METHOD M_Run
CASE _step OF
    0:
        M_Step(StepNo := 10, StepName := 'project.test.raiseIdle', Awaits := 0,
            AwaitingLabel := '', TimeClass := E_TimeClass.WORK, ExpectedTime := T#0S);
        _retVal := E_StepResult.ADVANCE;
        M_Advance(OnAdvance := 20);
    20:  // conditional command. `Enable` decides whether the child is driven at all,
         // so this step cannot hand it to the §6.9 auto-rollup - Awaits would name a
         // module it may never command. M_RaiseFromChild adopts the child's own
         // first-out instead, verbatim, with the child as the §3.13 drill-down link.
        M_Step(StepNo := 20, StepName := 'project.test.raiseCommand', Awaits := 0,
            AwaitingLabel := '', TimeClass := E_TimeClass.WORK, ExpectedTime := T#0S);
        IF ReportOnly THEN
            // The step already routes the failure itself, so it PUBLISHES the child's
            // first-out and carries on - the §6.9(e) counterpart of raising it.
            IF M_ReportFromChild(Source := _child) THEN
                _child.Execute := FALSE;
                _retVal := E_StepResult.ADVANCE;
            END_IF
        ELSIF M_RaiseFromChild(Source := _child) THEN
            _child.Execute := FALSE;         // §6.1 drop-reset frees the child to recover
            RETURN;                          // chain stopped; the Unit is in ERROR
        END_IF
        // §6.9(e) — called unconditionally every scan the step runs. The base
        // raises it ONCE per visit, so the ring gets one entry per occurrence and
        // the chain is never stopped by it.
        IF SimWarn THEN
            Warned := M_RaiseWarning(Reason := E_Reason.TEST_FAULT,
                DescriptionKey := 'project.test.stepWarning',
                Severity := E_Severity.LOW, Category := E_Category.PROCESS);
        END_IF
        IF Enable THEN
            IF M_TryIssue(Steppable := TRUE) THEN
                Issues := Issues + 1;        // proves the re-evaluation after resume
                _child.Abort := FALSE;
                _child.Execute := TRUE;
            END_IF
            IF _child.Done THEN
                _child.Execute := FALSE;
                _retVal := E_StepResult.ADVANCE;
            END_IF
        END_IF
        M_Advance(OnAdvance := 30);
    30:  // application rule: nothing in the framework can see it, so the step
         // defines the whole message - severity, category and drill-down link (§8.1).
        M_Step(StepNo := 30, StepName := 'project.test.raiseCustom', Awaits := 0,
            AwaitingLabel := '', TimeClass := E_TimeClass.WORK, ExpectedTime := T#0S);
        IF SimCustom THEN
            // A PROJECT BAND code (10000+), deliberately: M_RaiseCustom documents
            // that Severity/Category are a proposal the §8.8 rationalization
            // overrides for any REGISTERED reason, and every E_Reason member is
            // registered by construction (the catalog generator refuses one that
            // is not). Raising E_Reason.TEST_FAULT here therefore asserted the
            // opposite of what the test says it proves: the registry's LOW/SYSTEM
            // correctly replaced the step's HIGH/PROCESS. Only a band code the
            // registry does not know keeps the step's own choice.
            IF M_RaiseCustom(Reason := 10999,
                DescriptionKey := 'project.test.customRaise',
                Severity := E_Severity.HIGH, Category := E_Category.PROCESS,
                LinkPath := _child.Name) THEN
                RETURN;
            END_IF
        END_IF
        _retVal := E_StepResult.ADVANCE;
        M_Advance(OnAdvance := 999);
    999:
        M_Step(StepNo := 999, StepName := 'project.test.raiseComplete', Awaits := 0,
            AwaitingLabel := '', TimeClass := E_TimeClass.WORK, ExpectedTime := T#0S);
        Done := TRUE;
        M_Complete();
ELSE
    M_Fault(Reason := E_Reason.STEP_STALLED, DescriptionKey := 'std.error.undefinedStep');
END_CASE
END_METHOD

END_FUNCTION_BLOCK

// ---- Fraktal_Tests/FB_SequencePar_Tests.TcPOU
// Core §6.12 — parallel branches. Proves the three things that make them real
// rather than drawn: both legs run in the SAME scan with independent latches, the
// join waits for the slowest, and each leg is published as its own §3.13 rows.
FUNCTION_BLOCK FB_SequencePar_Tests EXTENDS TcUnit.FB_TestSuite
VAR
    _u : FB_ProbeUnitPar;
    _w1, _w2 : BOOL;
    _rowA, _rowB : INT;
    _i : INT;
END_VAR

Legs_run_together_with_independent_step_state();
Join_waits_for_every_leg_and_publishes_them_separately();

METHOD Legs_run_together_with_independent_step_state
TEST('Legs_run_together_with_independent_step_state');
IF NOT _w1 THEN
    AssertTrue(Condition := _u.Setup(Name := 'Test.Par'), Message := 'Unit sets up');
    AssertTrue(Condition := _u.Start(), Message := 'Unit starts');
    _u();                                // fork scan: BOTH legs run
    AssertEquals_UDINT(Expected := 1, Actual := _u.M_TestIssues(Leg := 1),
        Message := 'leg 1 issued its command');
    AssertEquals_UDINT(Expected := 1, Actual := _u.M_TestIssues(Leg := 2),
        Message := 'leg 2 issued its own command in the SAME scan - one shared issue latch used to let leg 1 consume the latch belonging to leg 2');
    _u();
    AssertEquals_UDINT(Expected := 1, Actual := _u.M_TestIssues(Leg := 1),
        Message := 'and neither re-issues while its step is still running (§6.1 one-shot, per leg)');
    _w1 := TRUE;
END_IF
TEST_FINISHED();
END_METHOD

METHOD Join_waits_for_every_leg_and_publishes_them_separately
TEST('Join_waits_for_every_leg_and_publishes_them_separately');
IF NOT _w2 THEN
    // both leg rows are live at once - the whole reason a single CurrentStep was
    // not enough to draw a parallel step (§3.13/§6.12)
    FOR _i := 1 TO _u.SequenceStepCount DO
        IF _u.SequenceStepDef[_i].StepNo = 600 THEN _rowA := _i; END_IF
        IF _u.SequenceStepDef[_i].StepNo = 700 THEN _rowB := _i; END_IF
    END_FOR
    AssertTrue(Condition := (_rowA > 0) AND (_rowB > 0),
        Message := 'each leg publishes its own rows, offset by its BaseStepNo');
    AssertEquals_INT(Expected := 1, Actual := _u.SequenceStepDef[_rowA].Branch,
        Message := 'tagged with the leg the fork assigned it');
    AssertEquals_INT(Expected := 2, Actual := _u.SequenceStepDef[_rowB].Branch,
        Message := 'and the other leg with its own');
    AssertTrue(Condition := (_u.ActiveSteps[1].RowIdx = _rowA)
        AND (_u.ActiveSteps[2].RowIdx = _rowB),
        Message := 'BOTH rows are active at the same time - one cursor per leg');
    // leg 1 finishes; the join must not fire on it alone
    _u.M_TestSetChild(Which := 1, ChildDone := TRUE);
    _u();                                // child A completes
    _u();                                // leg 1 advances to its terminal step
    _u();                                // leg 1 reports Done
    AssertEquals_INT(Expected := 500, Actual := _u.M_TestChainStep(),
        Message := 'the join holds the fork step while leg 2 is still working');
    AssertFalse(Condition := _u.Done, Message := 'and the Unit has not completed');
    _u.M_TestSetChild(Which := 2, ChildDone := TRUE);
    _u();                                // child B completes
    _u();                                // leg 2 advances
    _u();                                // leg 2 Done -> join fires
    _u();                                // chain reaches its completion step
    AssertEquals_INT(Expected := 999, Actual := _u.M_TestChainStep(),
        Message := 'the fork step commits only once EVERY leg is Done');
    _w2 := TRUE;
END_IF
TEST_FINISHED();
END_METHOD

END_FUNCTION_BLOCK

// ---- Fraktal_Tests/FB_ProbeUnitPar.TcPOU
// Unit host for the §6.12 parallel suite: two children, one forking chain.
FUNCTION_BLOCK FB_ProbeUnitPar EXTENDS FB_UnitBase
VAR
    ChildA : FB_ProbeCM;
    ChildB : FB_ProbeCM;
    Chain : FB_ProbeParChain;
END_VAR

Cyclic();

METHOD Setup : BOOL
VAR_INPUT
    Name : STRING(80);
END_VAR
_M_SetName(Name);
StallTime := T#10S;
Setup := ChildA.Setup(Name := CONCAT(Name, '.ChildA'))
    AND ChildB.Setup(Name := CONCAT(Name, '.ChildB'))
    AND _M_Register(Child := ChildA)
    AND _M_Register(Child := ChildB)
    AND Chain.Setup(Host := THIS^, ChildA := ChildA, ChildB := ChildB);
END_METHOD

METHOD PROTECTED OnCyclic : DINT
OnCyclic := SUPER^.OnCyclic();   // base first (Core §3.14.2)
_M_TickChildren();
END_METHOD

METHOD PROTECTED _M_Dispatch
Chain.M_Run();
END_METHOD

METHOD PROTECTED OnCommandStart : DINT
OnCommandStart := SUPER^.OnCommandStart();
Chain.M_Reset();
END_METHOD

METHOD M_TestSetChild : BOOL
VAR_INPUT
    Which : INT;
    ChildDone : BOOL;
END_VAR
IF Which = 1 THEN
    ChildA.SimDone := ChildDone;
ELSE
    ChildB.SimDone := ChildDone;
END_IF
M_TestSetChild := TRUE;
END_METHOD

METHOD M_TestIssues : UDINT
VAR_INPUT
    Leg : INT;
END_VAR
M_TestIssues := Chain.M_TestIssues(Leg := Leg);
END_METHOD

METHOD M_TestChainStep : INT
M_TestChainStep := Chain.ActiveStep;
END_METHOD

END_FUNCTION_BLOCK

// ---- Fraktal_Tests/FB_ProbeParChain.TcPOU
// §6.12 — the ST form of a parallel divergence: ONE fork step that runs each leg
// and joins on all of them. Two work positions running simultaneously and
// independently is exactly this shape, and it needs no chart.
FUNCTION_BLOCK FB_ProbeParChain EXTENDS FB_SequenceBase
VAR
    LegA : FB_ProbeLeg;
    LegB : FB_ProbeLeg;
END_VAR

;

METHOD Setup : BOOL
VAR_INPUT
    Host : I_SequenceHost;
END_VAR
VAR_IN_OUT
    ChildA : FB_ProbeCM;
    ChildB : FB_ProbeCM;
END_VAR
Setup := M_Attach(Host := Host)
    AND LegA.Setup(Host := Host, Child := ChildA)
    AND LegB.Setup(Host := Host, Child := ChildB);
END_METHOD

METHOD M_Reset
M_ResetBase(FirstStep := 0);
END_METHOD

METHOD M_Run
CASE _step OF
    0:  // the fork. One M_RunPar per leg, one M_ParJoin: the leg list is the calls
        // themselves, so there is nothing to register and nothing to keep in step
        // when a leg is added or removed (§1.1 O1).
        M_Step(StepNo := 500, StepName := 'project.test.forkBothPositions', Awaits := 0,
            AwaitingLabel := '', TimeClass := E_TimeClass.WORK, ExpectedTime := T#0S);
        M_RunPar(Chain := LegA, BaseStepNo := 600, Branch := 1);
        M_RunPar(Chain := LegB, BaseStepNo := 700, Branch := 2);
        _retVal := M_ParJoin();
        M_Advance(OnAdvance := 999);
    999:
        M_Step(StepNo := 999, StepName := 'project.test.parallelComplete', Awaits := 0,
            AwaitingLabel := '', TimeClass := E_TimeClass.WORK, ExpectedTime := T#0S);
        Done := TRUE;
        M_Complete();
ELSE
    M_Fault(Reason := E_Reason.STEP_STALLED, DescriptionKey := 'std.error.undefinedStep');
END_CASE
END_METHOD

// test seam: how many times each leg issued its own command
METHOD M_TestIssues : UDINT
VAR_INPUT
    Leg : INT;
END_VAR
IF Leg = 1 THEN
    M_TestIssues := LegA.Issues;
ELSE
    M_TestIssues := LegB.Issues;
END_IF
END_METHOD

END_FUNCTION_BLOCK

// ---- Fraktal_Tests/FB_ProbeLeg.TcPOU
// §6.12 — one leg of a parallel step, written as an ORDINARY chain. That is the
// whole point of the ST form: a leg is a chain, so it brings its own step pointer,
// its own transition result and its own step-scoped latches, and nothing about it
// has to know it is running beside another one.
FUNCTION_BLOCK FB_ProbeLeg EXTENDS FB_SequenceBase
VAR_OUTPUT
    Issues : UDINT;                    // times this leg issued its command
END_VAR
VAR
    {attribute 'OPC.UA.DA' := '0'}
    _child : REFERENCE TO FB_ProbeCM;
END_VAR

;

METHOD Setup : BOOL
VAR_INPUT
    Host : I_SequenceHost;
END_VAR
VAR_IN_OUT
    Child : FB_ProbeCM;
END_VAR
_child REF= Child;
Setup := M_Attach(Host := Host) AND __ISVALIDREF(_child);
END_METHOD

METHOD PROTECTED OnChainReset
Issues := 0;
END_METHOD

// Run as a composite/parallel leg, so the step records are offset by _baseStepNo
// (§6.5) and the chart still reads as one continuous chain.
METHOD M_ChainRun
CASE _step OF
    0:
        M_Step(StepNo := _baseStepNo, StepName := 'project.test.legCommand', Awaits := 0,
            AwaitingLabel := '', TimeClass := E_TimeClass.WORK, ExpectedTime := T#0S);
        IF M_TryIssue(Steppable := TRUE) THEN
            Issues := Issues + 1;
            _child.Abort := FALSE;
            _child.Execute := TRUE;
        END_IF
        IF _child.Done THEN
            _child.Execute := FALSE;
            _retVal := E_StepResult.ADVANCE;
        END_IF
        M_Advance(OnAdvance := 999);
    999:
        M_Step(StepNo := _baseStepNo + 90, StepName := 'project.test.legDone', Awaits := 0,
            AwaitingLabel := '', TimeClass := E_TimeClass.WORK, ExpectedTime := T#0S);
        Done := TRUE;                  // the join reads this
ELSE
    M_Fault(Reason := E_Reason.STEP_STALLED, DescriptionKey := 'std.error.undefinedStep');
END_CASE
END_METHOD

END_FUNCTION_BLOCK

// ---- Fraktal_Tests/FB_StateFlag_Tests.TcPOU
// Core §3.12 — derived state flags. The point of the mechanism is that a flag is
// a live fact, not a latch, so the tests are about what happens when the fact
// changes and when the module stops asserting it at all.
FUNCTION_BLOCK FB_StateFlag_Tests EXTENDS TcUnit.FB_TestSuite
VAR
    _m : FB_ProbeCM;
    _w1, _w2 : BOOL;
    _since : DT;
END_VAR

Flag_is_published_with_the_moment_it_changed();
Unpublished_flag_goes_stale_and_stops_claiming();

METHOD Flag_is_published_with_the_moment_it_changed
TEST('Flag_is_published_with_the_moment_it_changed');
IF NOT _w1 THEN
    AssertTrue(Condition := _m.Setup(Name := 'Test.State'), Message := 'module sets up');
    _m.SimState := TRUE;
    _m();
    AssertTrue(Condition := _m.StateProbe,
        Message := 'the call returns the value, so it reads as a plain assignment');
    AssertEquals_INT(Expected := 1, Actual := _m.StateFlagCount,
        Message := 'and publishes it on the generic table');
    AssertEquals_STRING(Expected := 'project.test.probeState',
        Actual := _m.StateFlags[1].Key, Message := 'under the key the module chose');
    AssertTrue(Condition := _m.StateFlags[1].Value, Message := 'with the value');
    AssertFalse(Condition := _m.StateFlags[1].Stale, Message := 'and not stale');
    _since := _m.StateFlags[1].Since;
    _m();
    AssertEquals_DWORD(Expected := DT_TO_DWORD(_since),
        Actual := DT_TO_DWORD(_m.StateFlags[1].Since),
        Message := 'Since is the moment it CHANGED, not the last time it was written');
    // the fact stops being true: a derived flag follows it with no sequence involved
    _m.SimState := FALSE;
    _m();
    AssertFalse(Condition := _m.StateFlags[1].Value,
        Message := 'a derived flag drops itself - this is what a latched OutCmd could not do');
    _w1 := TRUE;
END_IF
TEST_FINISHED();
END_METHOD

METHOD Unpublished_flag_goes_stale_and_stops_claiming
TEST('Unpublished_flag_goes_stale_and_stops_claiming');
IF NOT _w2 THEN
    _m.SimState := TRUE;
    _m();
    AssertTrue(Condition := _m.StateFlags[1].Value, Message := 'true again');
    // the project puts the publication behind a condition that stops being true
    _m.SimPublish := FALSE;
    _m();                                // last scan's publication still stands
    _m();                                // the sweep resolves it
    AssertTrue(Condition := _m.StateFlags[1].Stale,
        Message := 'a flag nobody computes any more is marked stale');
    AssertFalse(Condition := _m.StateFlags[1].Value,
        Message := 'and forced FALSE: unmaintained state is not a claim (§5.6)');
    _w2 := TRUE;
END_IF
TEST_FINISHED();
END_METHOD

END_FUNCTION_BLOCK

// ---- Fraktal_Tests/FB_Axis_Tests.TcPOU
// Annex G axis CM. T1/T4 are proven once in FB_Base_Tests and not repeated (S5.7).
//
// SCOPE, stated plainly: this host has no NC PTP licence, so no test here moves a
// real axis. Every test below asserts behaviour that occurs BEFORE any MC_* call
// is issued - request validation, the ownership contract, and the handshake. The
// MC_* interaction itself is unproven and recorded as such in the evidence.
//
// That is also why _M_MoveTo validates the request (soft limits) before the state
// (homed): both rejections are provable without a drive, and reporting "not
// homed" for an impossible target would send an operator to the wrong problem.
FUNCTION_BLOCK FB_Axis_Tests EXTENDS TcUnit.FB_TestSuite
VAR
    _ax1 : AXIS_REF;
    _cm1 : FB_AxisCM;
    _ax2 : AXIS_REF;
    _cm2 : FB_AxisCM;
    _ax3 : AXIS_REF;
    _cm3 : FB_AxisCM;
    _ax4 : AXIS_REF;
    _cm4 : FB_AxisCM;
    _w1, _w2, _w3, _w4 : BOOL;
END_VAR

Library_declares_no_interlocks_and_the_application_owns_safe_motion_status();
Target_outside_soft_limits_is_rejected_before_any_motion();
Move_before_home_is_rejected();
Unsupported_command_is_rejected();

METHOD Library_declares_no_interlocks_and_the_application_owns_safe_motion_status
TEST('Library_declares_no_interlocks_and_the_application_owns_safe_motion_status');
IF NOT _w1 THEN
    _cm1.Setup(Name := 'Axis1', AxisRef := _ax1, Recipe := 0);
    _cm1();
    // S7.2.1 + S9.2: a library cannot name "STO cleared" for a station it has
    // never seen, so it declares nothing and the application supplies the
    // read-only safe-motion status it can see.
    AssertTrue(Condition := _cm1.Intlk.AllOk,
        Message := 'a library type that declares no interlock does not gate the axis');
    AssertTrue(Condition := _cm1.DeclareCondition(Index := 1,
            DescriptionKey := 'std.interlock.areaSafe',
            Reason := E_Reason.INTERLOCK_DROPPED, Bypassable := FALSE),
        Message := 'the application declares its own safe-motion condition');
    _cm1();
    AssertFalse(Condition := _cm1.Intlk.AllOk,
        Message := 'a declared but undriven condition is fail-closed');
    _cm1.SetCondition(Index := 1, Ok := TRUE);
    _cm1();
    AssertTrue(Condition := _cm1.Intlk.AllOk, Message := 'and clears once driven');
    _w1 := TRUE;
END_IF
TEST_FINISHED();
END_METHOD

METHOD Target_outside_soft_limits_is_rejected_before_any_motion
TEST('Target_outside_soft_limits_is_rejected_before_any_motion');
IF NOT _w2 THEN
    _cm2.Setup(Name := 'Axis2', AxisRef := _ax2, Recipe := 0);
    _cm2.ParCfg.SoftMin := 0.0;
    _cm2.ParCfg.SoftMax := 100.0;
    _cm2.ParCmd.Target := 150.0;                  // beyond SoftMax
    _cm2.Command := E_AxisCommand.MOVE_TO;
    _cm2.Execute := TRUE;
    _cm2(); _cm2();
    // S5.6: reject the malformed request rather than commanding motion and
    // discovering the problem at a limit switch.
    AssertTrue(Condition := _cm2.Error, Message := 'an out-of-range target is refused');
    AssertEquals_DWORD(Expected := TO_DWORD(PL_ModuleReasons.AXIS_TARGET_OOR),
        Actual := _cm2.ErrorID, Message := 'with AXIS_TARGET_OOR');
    AssertEquals_STRING(Expected := 'Axis2', Actual := _cm2.Status.Diagnostic.SourcePath,
        Message := 'and the module as its source path');
    _w2 := TRUE;
END_IF
TEST_FINISHED();
END_METHOD

METHOD Move_before_home_is_rejected
TEST('Move_before_home_is_rejected');
IF NOT _w3 THEN
    _cm3.Setup(Name := 'Axis3', AxisRef := _ax3, Recipe := 0);
    _cm3.ParCfg.SoftMin := 0.0;
    _cm3.ParCfg.SoftMax := 100.0;
    _cm3.ParCmd.Target := 50.0;                   // in range, but the axis is not homed
    _cm3.Command := E_AxisCommand.MOVE_TO;
    _cm3.Execute := TRUE;
    _cm3(); _cm3();
    AssertTrue(Condition := _cm3.Error, Message := 'a move before homing is refused');
    AssertEquals_DWORD(Expected := TO_DWORD(PL_ModuleReasons.AXIS_NOT_HOMED),
        Actual := _cm3.ErrorID, Message := 'with AXIS_NOT_HOMED');
    AssertFalse(Condition := _cm3.OutImm.Homed, Message := 'and the axis reports not homed');
    _w3 := TRUE;
END_IF
TEST_FINISHED();
END_METHOD

METHOD Unsupported_command_is_rejected
TEST('Unsupported_command_is_rejected');
IF NOT _w4 THEN
    _cm4.Setup(Name := 'Axis4', AxisRef := _ax4, Recipe := 0);
    _cm4.Command := E_AxisCommand.NONE;           // never a valid request (S5.6)
    _cm4.Execute := TRUE;
    _cm4(); _cm4();
    AssertTrue(Condition := _cm4.Error, Message := 'an unset command is refused');
    AssertEquals_DWORD(Expected := TO_DWORD(E_Reason.UNSUPPORTED_COMMAND),
        Actual := _cm4.ErrorID, Message := 'with UNSUPPORTED_COMMAND');
    _w4 := TRUE;
END_IF
TEST_FINISHED();
END_METHOD

END_FUNCTION_BLOCK

// ---- Fraktal_Tests/FB_RobotPlanner_Tests.TcPOU
// Annex I I.9-I.10.2 route planner, against the geometry of the reviewed cell.
//
// The fixture is deliberately the real thing rather than a toy: five help
// points, the twelve work positions of a plasma-clean handling cell, and the
// scan position that sits between two transit regions - reachable from the
// drawer side via HELP4 and the process side via HELP5. That junction is the
// case the reference framework could not express declaratively and hand-coded
// in two different methods from private state; if the affinity table cannot
// reproduce it in BOTH directions with no branching, the model has failed and
// it is better to find out here than in an annex.
//
// No arm, no connector, no motion: the planner is pure logic (S5.7, Annex H).
FUNCTION_BLOCK FB_RobotPlanner_Tests EXTENDS TcUnit.FB_TestSuite
VAR CONSTANT
    // helps
    HELP1 : INT := 1;   // change-position side
    HELP2 : INT := 2;   // left drawer
    HELP3 : INT := 3;   // home / NIO drawer
    HELP4 : INT := 4;   // drawer-side scan approach
    HELP5 : INT := 5;   // process side
    // nests
    CP_GRIPPER1    : INT := 1;
    READ_GRIPPER   : INT := 2;
    SCAN_PART      : INT := 3;
    DRAWER_LEFT    : INT := 4;
    DRAWER_RIGHT   : INT := 5;
    DRAWER_NIO     : INT := 6;
    PROCESS_START  : INT := 7;
    ONE_WAY_NEST   : INT := 8;   // synthetic: entry-only, to prove the loud refusal
    ISLAND_NEST    : INT := 9;   // synthetic: served by a help with no graph edge
    // transit regions
    REGION_DRAWER  : DWORD := 1;
    REGION_PROCESS : DWORD := 2;
    // grippers
    G_WITH : INT := 1;   // a gripper is coupled - tall approach
    G_NONE : INT := 2;   // nothing coupled - short approach
END_VAR
VAR
    _graph : ST_RouteGraph;
    _geom  : ST_RobotGeometry;
    _p     : FB_RobotRoutePlanner;
    _route : ST_RobotPointList;
    _ret   : DINT;
    _help  : INT;
    _built : BOOL;
    _w1, _w2, _w3, _w4, _w5, _w6, _w7, _w8, _w9, _w10 : BOOL;
END_VAR

IF NOT _built THEN
    _M_BuildFixture();
    _built := TRUE;
END_IF

Scan_junction_resolves_the_process_side_help();
Scan_junction_resolves_the_drawer_side_help_in_the_same_table();
Nest_to_nest_emits_depart_then_transit_then_approach();
Approach_corridor_is_reversed_and_lands_exactly_on_the_nest();
Corridor_differs_per_gripper_with_no_conditional_code();
Taught_corridor_emits_a_list_reference_instead_of_offsets();
Disconnected_graph_yields_ROBOT_NO_ROUTE();
One_way_nest_refuses_the_reversal_loudly();
Malformed_endpoints_are_rejected_before_planning();
Direct_nest_list_bypasses_help_routing();

// The reviewed cell as configuration - which is the whole point: a station
// supplies a table, not traversal code.
METHOD PRIVATE _M_BuildFixture
VAR
    _i : INT;
END_VAR
// --- help geometry and the transit graph -------------------------------
_geom.HelpPose[HELP1].X := 0;    _geom.HelpPose[HELP1].Z := 1000;
_geom.HelpPose[HELP2].X := 500;  _geom.HelpPose[HELP2].Z := 1000;
_geom.HelpPose[HELP3].X := 1000; _geom.HelpPose[HELP3].Z := 1000;
_geom.HelpPose[HELP4].X := 1500; _geom.HelpPose[HELP4].Z := 1000;
_geom.HelpPose[HELP5].X := 2000; _geom.HelpPose[HELP5].Z := 1000;

_graph.HelpRegion[HELP1] := REGION_DRAWER;
_graph.HelpRegion[HELP2] := REGION_DRAWER;
_graph.HelpRegion[HELP3] := REGION_DRAWER;
_graph.HelpRegion[HELP4] := REGION_DRAWER;
_graph.HelpRegion[HELP5] := REGION_PROCESS;

// a simple chain HELP1..HELP5, bidirectional
FOR _i := 1 TO 4 DO
    _graph.HelpAdj[_i, _i + 1] := TRUE;
    _graph.HelpAdj[_i + 1, _i] := TRUE;
END_FOR

// --- nest geometry -----------------------------------------------------
_geom.NestPose[G_WITH, DRAWER_LEFT].X  := 500;
_geom.NestPose[G_WITH, DRAWER_LEFT].Y  := 200;
_geom.NestPose[G_WITH, DRAWER_LEFT].Z  := 100;
_geom.NestPose[G_NONE, DRAWER_LEFT]    := _geom.NestPose[G_WITH, DRAWER_LEFT];
_geom.NestPose[G_WITH, PROCESS_START].X := 2000;
_geom.NestPose[G_WITH, PROCESS_START].Z := 300;
_geom.NestPose[G_WITH, SCAN_PART].X     := 1500;
_geom.NestPose[G_WITH, SCAN_PART].Z     := 400;
_geom.NestPose[G_WITH, READ_GRIPPER].X  := 0;
_geom.NestPose[G_WITH, READ_GRIPPER].Z  := 200;

// --- affinity: single-help nests are the trivial case ------------------
_M_Affinity1(G_WITH, CP_GRIPPER1,   HELP1);
_M_Affinity1(G_WITH, READ_GRIPPER,  HELP1);
_M_Affinity1(G_WITH, DRAWER_LEFT,   HELP2);
_M_Affinity1(G_WITH, DRAWER_RIGHT,  HELP4);
_M_Affinity1(G_WITH, DRAWER_NIO,    HELP3);
_M_Affinity1(G_WITH, PROCESS_START, HELP5);
_M_Affinity1(G_NONE, DRAWER_LEFT,   HELP2);

// --- the junction: TWO corridors, both bidirectional, split by region ---
// This is the case the reference hand-codes. Here it is two table rows.
_graph.NestHelp[G_WITH, SCAN_PART].Count := 2;
_graph.NestHelp[G_WITH, SCAN_PART].Helps[1].HelpId   := HELP4;
_graph.NestHelp[G_WITH, SCAN_PART].Helps[1].Role     := E_HelpRole.EITHER;
_graph.NestHelp[G_WITH, SCAN_PART].Helps[1].RegionId := REGION_DRAWER;
_graph.NestHelp[G_WITH, SCAN_PART].Helps[2].HelpId   := HELP5;
_graph.NestHelp[G_WITH, SCAN_PART].Helps[2].Role     := E_HelpRole.EITHER;
_graph.NestHelp[G_WITH, SCAN_PART].Helps[2].RegionId := REGION_PROCESS;

// --- a genuinely one-way nest: entry only ------------------------------
_graph.NestHelp[G_WITH, ONE_WAY_NEST].Count := 1;
_graph.NestHelp[G_WITH, ONE_WAY_NEST].Helps[1].HelpId := HELP3;
_graph.NestHelp[G_WITH, ONE_WAY_NEST].Helps[1].Role   := E_HelpRole.APPROACH;

// --- a nest whose help has no edge into the graph -----------------------
_graph.NestHelp[G_WITH, ISLAND_NEST].Count := 1;
_graph.NestHelp[G_WITH, ISLAND_NEST].Helps[1].HelpId := 7;   // HelpAdj[7,*] all FALSE

// --- corridors: the reference's real geometry --------------------------
// With a gripper coupled the arm backs out and lifts; with nothing coupled it
// simply clears. Same nest, different gripper index - no conditional code.
_M_Corridor2(G_WITH, DRAWER_LEFT, HELP2, 0, -100, 0, 0, -100, 200);
_M_Corridor1(G_NONE, DRAWER_LEFT, HELP2, 0, 0, 50);
END_METHOD

// One nest served by one help, both directions, offsets unset.
METHOD PRIVATE _M_Affinity1
VAR_INPUT
    Gripper : INT;
    Nest    : INT;
    HelpId  : INT;
END_VAR
_graph.NestHelp[Gripper, Nest].Count := 1;
_graph.NestHelp[Gripper, Nest].Helps[1].HelpId := HelpId;
_graph.NestHelp[Gripper, Nest].Helps[1].Role   := E_HelpRole.EITHER;
END_METHOD

// A one-step corridor, used for both approach and depart.
METHOD PRIVATE _M_Corridor1
VAR_INPUT
    Gripper : INT;
    Nest    : INT;
    HelpId  : INT;
    DX, DY, DZ : LREAL;
END_VAR
VAR
    _i : INT;
END_VAR
_i := _M_FindAffinity(Gripper, Nest, HelpId);
IF _i = 0 THEN RETURN; END_IF
_graph.NestHelp[Gripper, Nest].Helps[_i].Approach.StepCount := 1;
_graph.NestHelp[Gripper, Nest].Helps[_i].Approach.Steps[1].D.X := DX;
_graph.NestHelp[Gripper, Nest].Helps[_i].Approach.Steps[1].D.Y := DY;
_graph.NestHelp[Gripper, Nest].Helps[_i].Approach.Steps[1].D.Z := DZ;
_graph.NestHelp[Gripper, Nest].Helps[_i].Approach.Steps[1].MoveClass := E_MoveClass.SLOW_LINEAR;
_graph.NestHelp[Gripper, Nest].Helps[_i].Depart := _graph.NestHelp[Gripper, Nest].Helps[_i].Approach;
END_METHOD

// A two-step corridor - the reference's "back out, then lift" retract.
METHOD PRIVATE _M_Corridor2
VAR_INPUT
    Gripper : INT;
    Nest    : INT;
    HelpId  : INT;
    D1X, D1Y, D1Z : LREAL;
    D2X, D2Y, D2Z : LREAL;
END_VAR
VAR
    _i : INT;
END_VAR
_i := _M_FindAffinity(Gripper, Nest, HelpId);
IF _i = 0 THEN RETURN; END_IF
_graph.NestHelp[Gripper, Nest].Helps[_i].Approach.StepCount := 2;
_graph.NestHelp[Gripper, Nest].Helps[_i].Approach.Steps[1].D.X := D1X;
_graph.NestHelp[Gripper, Nest].Helps[_i].Approach.Steps[1].D.Y := D1Y;
_graph.NestHelp[Gripper, Nest].Helps[_i].Approach.Steps[1].D.Z := D1Z;
_graph.NestHelp[Gripper, Nest].Helps[_i].Approach.Steps[1].MoveClass := E_MoveClass.SLOW_LINEAR;
_graph.NestHelp[Gripper, Nest].Helps[_i].Approach.Steps[2].D.X := D2X;
_graph.NestHelp[Gripper, Nest].Helps[_i].Approach.Steps[2].D.Y := D2Y;
_graph.NestHelp[Gripper, Nest].Helps[_i].Approach.Steps[2].D.Z := D2Z;
_graph.NestHelp[Gripper, Nest].Helps[_i].Approach.Steps[2].MoveClass := E_MoveClass.SLOW_LINEAR;
_graph.NestHelp[Gripper, Nest].Helps[_i].Depart := _graph.NestHelp[Gripper, Nest].Helps[_i].Approach;
END_METHOD

METHOD PRIVATE _M_FindAffinity : INT
VAR_INPUT
    Gripper : INT;
    Nest    : INT;
    HelpId  : INT;
END_VAR
VAR
    _i : INT;
END_VAR
_M_FindAffinity := 0;
FOR _i := 1 TO _graph.NestHelp[Gripper, Nest].Count DO
    IF _graph.NestHelp[Gripper, Nest].Helps[_i].HelpId = HelpId THEN
        _M_FindAffinity := _i;
        RETURN;
    END_IF
END_FOR
END_METHOD

METHOD PRIVATE Scan_junction_resolves_the_process_side_help
TEST('Scan_junction_resolves_the_process_side_help');
IF NOT _w1 THEN
    _p.rGraph REF= _graph;
    _p.rGeom  REF= _geom;
    // Leaving the scan position toward PROCESS_START. Both corridors are
    // bidirectional, so the direction filter keeps both and the REGION of the
    // other endpoint decides - reproducing the reference's hand-coded choice.
    _help := _p.ResolveHelp(Gripper := G_WITH, Nest := SCAN_PART,
        OtherRegion := REGION_PROCESS, Dir := E_HelpRole.DEPART);
    AssertEquals_INT(Expected := HELP5, Actual := _help,
        Message := 'a move toward the process side leaves scan via HELP5');
    _w1 := TRUE;
END_IF
TEST_FINISHED();
END_METHOD

METHOD PRIVATE Scan_junction_resolves_the_drawer_side_help_in_the_same_table
TEST('Scan_junction_resolves_the_drawer_side_help_in_the_same_table');
IF NOT _w2 THEN
    _p.rGraph REF= _graph;
    _p.rGeom  REF= _geom;
    // Same two table rows, opposite direction, no per-direction duplication -
    // which is exactly what the reference needed two hand-written methods for.
    _help := _p.ResolveHelp(Gripper := G_WITH, Nest := SCAN_PART,
        OtherRegion := REGION_DRAWER, Dir := E_HelpRole.APPROACH);
    AssertEquals_INT(Expected := HELP4, Actual := _help,
        Message := 'a move from the drawer side enters scan via HELP4');
    _w2 := TRUE;
END_IF
TEST_FINISHED();
END_METHOD

METHOD PRIVATE Nest_to_nest_emits_depart_then_transit_then_approach
TEST('Nest_to_nest_emits_depart_then_transit_then_approach');
IF NOT _w3 THEN
    _p.rGraph REF= _graph;
    _p.rGeom  REF= _geom;
    _ret := _p.BuildRoute(Gripper := G_WITH, FromNest := DRAWER_LEFT, FromHelp := 0,
        ToNest := 0, ToHelp := HELP5, Route := _route);
    AssertEquals_DINT(Expected := 0, Actual := _ret,
        Message := 'a routable pair plans without error');
    // 2 depart offsets + the help chain HELP2,HELP3,HELP4,HELP5
    AssertEquals_INT(Expected := 6, Actual := _route.Count,
        Message := 'depart corridor then the transit chain');
    AssertTrue(Condition := _route.Points[1].MoveClass = E_MoveClass.SLOW_LINEAR,
        Message := 'pre-positions are flown slow');
    AssertTrue(Condition := _route.Points[3].MoveClass = E_MoveClass.FAST_PTP,
        Message := 'transit between helps is flown fast');
    AssertEquals_LREAL(Expected := 2000, Actual := _route.Points[6].Target.X, Delta := 0.001,
        Message := 'and it ends on the target help');
    _w3 := TRUE;
END_IF
TEST_FINISHED();
END_METHOD

METHOD PRIVATE Approach_corridor_is_reversed_and_lands_exactly_on_the_nest
TEST('Approach_corridor_is_reversed_and_lands_exactly_on_the_nest');
IF NOT _w4 THEN
    _p.rGraph REF= _graph;
    _p.rGeom  REF= _geom;
    _ret := _p.BuildRoute(Gripper := G_WITH, FromNest := 0, FromHelp := HELP5,
        ToNest := DRAWER_LEFT, ToHelp := 0, Route := _route);
    AssertEquals_DINT(Expected := 0, Actual := _ret, Message := 'plans without error');
    // chain HELP5..HELP2 (4) + 2 approach offsets reversed + the nest itself
    AssertEquals_INT(Expected := 7, Actual := _route.Count,
        Message := 'transit chain, reversed approach, then the nest');
    // reversed: the FAR offset (-100,+200) is flown before the NEAR one (-100,0)
    AssertEquals_LREAL(Expected := 300, Actual := _route.Points[5].Target.Z, Delta := 0.001,
        Message := 'the outer pre-position comes first on the way in');
    AssertEquals_LREAL(Expected := 100, Actual := _route.Points[6].Target.Z, Delta := 0.001,
        Message := 'then the inner one');
    // S I.8: the last point of a path is reached exactly, never blended short
    AssertEquals_LREAL(Expected := 200, Actual := _route.Points[7].Target.Y, Delta := 0.001,
        Message := 'and the route lands exactly on the taught nest');
    AssertTrue(Condition := _route.Points[7].MoveClass = E_MoveClass.SLOW_LINEAR,
        Message := 'the final approach is linear, not blended PTP');
    _w4 := TRUE;
END_IF
TEST_FINISHED();
END_METHOD

METHOD PRIVATE Corridor_differs_per_gripper_with_no_conditional_code
TEST('Corridor_differs_per_gripper_with_no_conditional_code');
IF NOT _w5 THEN
    _p.rGraph REF= _graph;
    _p.rGeom  REF= _geom;
    // The reference branches on the clutch to pick a tall or short approach.
    // Affinity is indexed [gripper, nest], so the two are simply different
    // gripper indices - the state-dependence falls out of a dimension the
    // model already has (I.10.2).
    _ret := _p.BuildRoute(Gripper := G_NONE, FromNest := 0, FromHelp := HELP2,
        ToNest := DRAWER_LEFT, ToHelp := 0, Route := _route);
    AssertEquals_DINT(Expected := 0, Actual := _ret, Message := 'plans without error');
    // HELP2 only (start = target help) + 1 approach offset + the nest
    AssertEquals_INT(Expected := 3, Actual := _route.Count,
        Message := 'with nothing coupled the short corridor is one step');
    AssertEquals_LREAL(Expected := 150, Actual := _route.Points[2].Target.Z, Delta := 0.001,
        Message := 'clearing by 50 rather than lifting by 200');
    _w5 := TRUE;
END_IF
TEST_FINISHED();
END_METHOD

METHOD PRIVATE Taught_corridor_emits_a_list_reference_instead_of_offsets
VAR
    _i : INT;
END_VAR
TEST('Taught_corridor_emits_a_list_reference_instead_of_offsets');
IF NOT _w6 THEN
    _p.rGraph REF= _graph;
    _p.rGeom  REF= _geom;
    // Generation is the default, teaching the escape hatch: StepCount = 0 with
    // a ListId names a taught list for geometry offsets cannot express (I.10.2).
    _i := _M_FindAffinity(G_WITH, READ_GRIPPER, HELP1);
    _graph.NestHelp[G_WITH, READ_GRIPPER].Helps[_i].Approach.StepCount := 0;
    _graph.NestHelp[G_WITH, READ_GRIPPER].Helps[_i].Approach.ListId    := 77;
    _ret := _p.BuildRoute(Gripper := G_WITH, FromNest := 0, FromHelp := HELP1,
        ToNest := READ_GRIPPER, ToHelp := 0, Route := _route);
    AssertEquals_DINT(Expected := 0, Actual := _ret, Message := 'plans without error');
    AssertEquals_DWORD(Expected := 77, Actual := _route.Points[_route.Count].ListId,
        Message := 'the taught list is named for the executor to run');
    _w6 := TRUE;
END_IF
TEST_FINISHED();
END_METHOD

METHOD PRIVATE Disconnected_graph_yields_ROBOT_NO_ROUTE
TEST('Disconnected_graph_yields_ROBOT_NO_ROUTE');
IF NOT _w7 THEN
    _p.rGraph REF= _graph;
    _p.rGeom  REF= _geom;
    // ISLAND_NEST's serving help has no edge into the transit graph. The
    // planner refuses with a clean first-out rather than inventing a move.
    _ret := _p.BuildRoute(Gripper := G_WITH, FromNest := 0, FromHelp := HELP1,
        ToNest := ISLAND_NEST, ToHelp := 0, Route := _route);
    AssertEquals_DINT(Expected := PL_ModuleReasons.ROBOT_NO_ROUTE, Actual := _ret,
        Message := 'an unreachable help is ROBOT_NO_ROUTE, not a silent move');
    AssertEquals_INT(Expected := 0, Actual := _route.Count,
        Message := 'and no partial route is left behind');
    _w7 := TRUE;
END_IF
TEST_FINISHED();
END_METHOD

METHOD PRIVATE One_way_nest_refuses_the_reversal_loudly
TEST('One_way_nest_refuses_the_reversal_loudly');
IF NOT _w8 THEN
    _p.rGraph REF= _graph;
    _p.rGeom  REF= _geom;
    // Entry is legal...
    _help := _p.ResolveHelp(Gripper := G_WITH, Nest := ONE_WAY_NEST,
        OtherRegion := 0, Dir := E_HelpRole.APPROACH);
    AssertEquals_INT(Expected := HELP3, Actual := _help,
        Message := 'an APPROACH-only nest can be entered');
    // ...and leaving through it is refused rather than mis-routed. This is the
    // NOK-reversal case of I.10.1: a real cell constraint surfaced, loudly.
    _ret := _p.BuildRoute(Gripper := G_WITH, FromNest := ONE_WAY_NEST, FromHelp := 0,
        ToNest := 0, ToHelp := HELP1, Route := _route);
    AssertEquals_DINT(Expected := PL_ModuleReasons.ROBOT_NO_HELP_FOR_NEST, Actual := _ret,
        Message := 'and reversing out of it fails loudly, never silently');
    _w8 := TRUE;
END_IF
TEST_FINISHED();
END_METHOD

METHOD PRIVATE Malformed_endpoints_are_rejected_before_planning
TEST('Malformed_endpoints_are_rejected_before_planning');
IF NOT _w9 THEN
    _p.rGraph REF= _graph;
    _p.rGeom  REF= _geom;
    // Both a nest AND a help at one end is malformed regardless of geometry,
    // so it is rejected before anything is resolved (S5.6).
    _ret := _p.BuildRoute(Gripper := G_WITH, FromNest := DRAWER_LEFT, FromHelp := HELP2,
        ToNest := 0, ToHelp := HELP5, Route := _route);
    AssertTrue(Condition := _ret <> 0,
        Message := 'a start that is both a nest and a help is refused');
    // Neither is equally malformed.
    _ret := _p.BuildRoute(Gripper := G_WITH, FromNest := 0, FromHelp := HELP2,
        ToNest := 0, ToHelp := 0, Route := _route);
    AssertTrue(Condition := _ret <> 0, Message := 'and so is a target that is neither');
    _w9 := TRUE;
END_IF
TEST_FINISHED();
END_METHOD

METHOD PRIVATE Direct_nest_list_bypasses_help_routing
TEST('Direct_nest_list_bypasses_help_routing');
IF NOT _w10 THEN
    _p.rGraph REF= _graph;
    _p.rGeom  REF= _geom;
    _graph.DirectNest[DRAWER_LEFT, PROCESS_START] := 42;
    _ret := _p.BuildRoute(Gripper := G_WITH, FromNest := DRAWER_LEFT, FromHelp := 0,
        ToNest := PROCESS_START, ToHelp := 0, Route := _route);
    AssertEquals_DINT(Expected := 0, Actual := _ret, Message := 'plans without error');
    AssertEquals_INT(Expected := 1, Actual := _route.Count,
        Message := 'a taught direct list replaces the whole generated route');
    AssertEquals_DWORD(Expected := 42, Actual := _route.Points[1].ListId,
        Message := 'and names that list');
    _graph.DirectNest[DRAWER_LEFT, PROCESS_START] := 0;
    _w10 := TRUE;
END_IF
TEST_FINISHED();
END_METHOD

END_FUNCTION_BLOCK

// ---- Fraktal_Tests/FB_RobotConnector_Tests.TcPOU
// Annex I I.3/I.5 - the Staubli VAL3 connector over the SIM channel. No socket,
// no emulator, no arm: FB_SimByteChannel scripts request/reply pairs, so the wire
// protocol and every refusal path are provable in CI (S5.7, Annex H).
//
// This is the transport-layer half of the I.5c simulation requirement. The SRS
// Emulator remains the higher-fidelity layer for motion behaviour; what is proven
// here is the part that must hold before an emulator is worth starting: that the
// connector speaks the agreed frames, and that it REFUSES rather than pretends
// when the link is down, the mode is wrong, or the path was left.
//
// Linked means session up AND heartbeat healthy (Core §3.15.2), and the heartbeat
// is the TON-driven status poll, so every test that needs a live link runs ACROSS
// SCANS and scripts the STA reply the heartbeat asks for.
FUNCTION_BLOCK FB_RobotConnector_Tests EXTENDS TcUnit.FB_TestSuite
VAR
    _chan  : FB_SimByteChannel;
    _conn  : FB_StaubliVal3Connector;
    _chanB : FB_SimByteChannel;
    _connB : FB_StaubliVal3Connector;
    _chanC : FB_SimByteChannel;
    _connC : FB_StaubliVal3Connector;
    _chanD : FB_SimByteChannel;
    _connD : FB_StaubliVal3Connector;
    _ok    : BOOL;
    _i, _i2, _i4 : INT;
    _diag  : ST_Diagnostic;   // C0185: cannot access .member on a property result
    _pose  : ST_RobotPose;
    _w1, _w2, _w3, _w4, _w5, _w6 : BOOL;
    _sent2, _sent4 : BOOL;
END_VAR

Link_down_refuses_every_command_rather_than_dropping_it();
Id_addressed_commands_are_framed_on_the_wire();
Status_poll_publishes_the_controllers_reported_facts();
Controller_error_is_carried_verbatim_and_faults();
Resume_is_refused_when_the_arm_left_the_retained_path();
Unknown_mode_request_is_refused_outright();

METHOD PRIVATE Link_down_refuses_every_command_rather_than_dropping_it
TEST('Link_down_refuses_every_command_rather_than_dropping_it');
IF NOT _w1 THEN
    // Deliberately never set up or connected: there is no session.
    // A command issued now must come back FALSE. Silently queueing it would let a
    // sequence wait on a robot that never heard the command (Annex D).
    AssertFalse(Condition := _connB.PowerOn(),
        Message := 'a command on a down link is refused, not queued');
    AssertFalse(Condition := _connB.MoveToPoint(PointId := 7),
        Message := 'and so is an ID-addressed move');
    AssertFalse(Condition := _connB.Linked,
        Message := 'Linked reports the link honestly');
    _diag := _connB.LastResult;
    AssertEquals_DINT(Expected := E_Reason.LINK_TIMEOUT, Actual := _diag.ReasonCode,
        Message := 'the refusal carries the link reason for the CM to adopt');
    _w1 := TRUE;
END_IF
TEST_FINISHED();
END_METHOD

METHOD PRIVATE Id_addressed_commands_are_framed_on_the_wire
TEST('Id_addressed_commands_are_framed_on_the_wire');
IF _w2 THEN
    TEST_FINISHED();
    RETURN;
END_IF
IF _i2 = 0 THEN
    // The channel only replies when the sent line matches EXACTLY, so a reply
    // proves the frame. Every argument is an identifier - never a coordinate (I.1).
    _chan.Script(Expect := 'STA$R', Reply := 'STA,OK,0,1,AUTO,4,0,1,0,0,0,0,0,0$R');
    _chan.Script(Expect := 'TPL,11,22$R', Reply := 'TPL,OK$R');
    _conn.SetupLink(Name := 'Test.Robot', Chan := _chan, DevHost := '10.0.0.20', DevPort := 11000);
    _conn.Connect();
END_IF
_conn.Cyclic();
_i2 := _i2 + 1;
IF _conn.Linked AND NOT _sent2 THEN
    AssertTrue(Condition := _conn.MoveTemplate(FromPosId := 11, ToPosId := 22),
        Message := 'a routed move is accepted and framed as TPL,from,to');
    _sent2 := TRUE;
ELSIF _sent2 AND (_conn.LastResponse = 'TPL,OK') THEN
    AssertEquals_STRING(Expected := 'TPL,OK', Actual := _conn.LastResponse,
        Message := 'and the controller acknowledgement is published');
    _w2 := TRUE;
    TEST_FINISHED();
ELSIF _i2 > 1000 THEN
    AssertTrue(Condition := FALSE,
        Message := 'the link never came up, or the framed move was never acknowledged');
    _w2 := TRUE;
    TEST_FINISHED();
END_IF
END_METHOD

METHOD PRIVATE Status_poll_publishes_the_controllers_reported_facts
TEST('Status_poll_publishes_the_controllers_reported_facts');
// The poll is the TON-driven heartbeat, so this test must run ACROSS SCANS - a loop
// of Cyclic() calls inside one scan advances no time and the timer never fires.
// Same shape as FB_TcpDev_Tests.Timeout_faults_10402, for the same reason.
IF _w3 THEN
    TEST_FINISHED();
    RETURN;
END_IF
IF _i = 0 THEN
    // STA,OK,busy,ref,mode,area,prot,resumable,x,y,z,rx,ry,rz
    _chanC.Script(Expect := 'STA$R',
        Reply := 'STA,OK,0,1,AUTO,4,0,1,100.5,200,300,0,0,90$R');
    _connC.SetupLink(Name := 'Test.RobotC', Chan := _chanC, DevHost := '10.0.0.21', DevPort := 11000);
    _connC.Connect();
END_IF
_connC.Cyclic();
_i := _i + 1;

IF _connC.Referenced THEN
    // Referenced only becomes TRUE once a status reply was parsed, so reaching
    // here proves the heartbeat fired, framed STA, and the reply was decoded.
    AssertTrue(Condition := _connC.Linked,
        Message := 'an answered status poll is a healthy heartbeat: the link is up');
    AssertTrue(Condition := _connC.ActualMode = E_RobotOpMode.AUTO_REMOTE,
        Message := 'ActualMode is what the controller REPORTS, not what we asked for');
    AssertEquals_DWORD(Expected := 4, Actual := _connC.CurrentArea,
        Message := 'the planning area is published for area-resolved motion');
    AssertFalse(Condition := _connC.ProtectiveStop,
        Message := 'the protective stop is published separately from S9 safety');
    _pose := _connC.ActualPosition;
    AssertEquals_LREAL(Expected := 100.5, Actual := _pose.X, Delta := 0.001,
        Message := 'the live pose is readable for display and diagnostics');
    AssertEquals_LREAL(Expected := 90, Actual := _pose.RZ, Delta := 0.001,
        Message := 'including orientation');
    // Jogging is bounded by the CONTROLLER's mode, not by a PLC release alone.
    // Asserted here because this is where a LINKED connector reporting AUTO
    // exists - proving the refusal comes from the mode gate and not the link.
    AssertFalse(Condition := _connC.Jog(Mode := E_RobotJogMode.JOINT, Axis := 1, Dir := 1),
        Message := 'jogging is refused while the controller reports auto');
    _w3 := TRUE;
    TEST_FINISHED();
ELSIF _i > 1000 THEN
    // Bounded so a regression fails loudly here instead of hanging the runner
    // with no message, which is the worse failure.
    AssertTrue(Condition := FALSE,
        Message := 'the status poll never delivered a reply');
    _w3 := TRUE;
    TEST_FINISHED();
END_IF
END_METHOD

METHOD PRIVATE Controller_error_is_carried_verbatim_and_faults
TEST('Controller_error_is_carried_verbatim_and_faults');
IF _w4 THEN
    TEST_FINISHED();
    RETURN;
END_IF
IF _i4 = 0 THEN
    _chanD.Script(Expect := 'STA$R', Reply := 'STA,OK,0,0,AUTO,0,0,0,0,0,0,0,0,0$R');
    _chanD.Script(Expect := 'HOME$R', Reply := 'HOME,ERR,J12,joint 3 out of range$R');
    _connD.SetupLink(Name := 'Test.RobotD', Chan := _chanD, DevHost := '10.0.0.22', DevPort := 11000);
    _connD.Connect();
END_IF
_connD.Cyclic();
_i4 := _i4 + 1;
_diag := _connD.ControllerMessage;
IF _connD.Linked AND NOT _sent4 THEN
    AssertTrue(Condition := _connD.Home(), Message := 'the request is accepted by the transport');
    _sent4 := TRUE;
ELSIF _sent4 AND (_diag.ReasonCode = PL_ModuleReasons.ROBOT_CONTROLLER_FAULT) THEN
    // The robot's OWN text survives. Paraphrasing it would cost the technician the
    // one string that identifies the fault on the pendant (S8.2).
    AssertTrue(Condition := FIND(_diag.Description, 'joint 3 out of range') > 0,
        Message := 'the controller message is carried verbatim');
    _diag := _connD.LastResult;
    AssertEquals_DINT(Expected := PL_ModuleReasons.ROBOT_CONTROLLER_FAULT,
        Actual := _diag.ReasonCode,
        Message := 'and it is the refusal the robot CM adopts as its first-out');
    AssertFalse(Condition := _connD.MotionBusy,
        Message := 'a refused command does not leave the connector claiming motion');
    _w4 := TRUE;
    TEST_FINISHED();
ELSIF _i4 > 1000 THEN
    AssertTrue(Condition := FALSE,
        Message := 'the controller error never arrived');
    _w4 := TRUE;
    TEST_FINISHED();
END_IF
END_METHOD

METHOD PRIVATE Resume_is_refused_when_the_arm_left_the_retained_path
TEST('Resume_is_refused_when_the_arm_left_the_retained_path');
IF NOT _w5 THEN
    // Resumable=0 in the status reply. A hold is exactly when an operator jogs the
    // arm, and resuming onto a path the tool has left is how a robot drives through
    // a fixture - so this must refuse rather than execute (I.4b).
    AssertFalse(Condition := _connD.Resumable,
        Message := 'the connector reports resumption invalid by default');
    AssertFalse(Condition := _connD.Resume(),
        Message := 'and Resume is refused rather than sent');
    _w5 := TRUE;
END_IF
TEST_FINISHED();
END_METHOD

METHOD PRIVATE Unknown_mode_request_is_refused_outright
TEST('Unknown_mode_request_is_refused_outright');
IF NOT _w6 THEN
    // Requesting UNKNOWN is meaningless and must never reach the controller: an
    // uninitialised or unparsed mode must not travel as though it were a real
    // request. Self-contained on purpose - the previous version asserted a
    // precondition owned by another test, so one root cause failed two tests.
    AssertFalse(Condition := _connB.RequestMode(Mode := E_RobotOpMode.UNKNOWN),
        Message := 'an UNKNOWN mode request is refused before the transport');
    _w6 := TRUE;
END_IF
TEST_FINISHED();
END_METHOD

END_FUNCTION_BLOCK

// ---- Fraktal_Tests/FB_RobotCM_Tests.TcPOU
// Annex I I.14 - the robot CM proven against the SIMULATED connector (I.5c).
// No arm, no emulator, no socket: FB_SimRobotConnector honours the handshake and
// injects the I.2 reasons on demand, which is the only way to prove refusals that
// would otherwise require deliberately breaking a cell.
//
// What is under test here is the CM's own contract - the S5.6 validation ladder,
// the S6.1 HELD translation, and the S8.2 rule that a connector's reason is
// ADOPTED rather than re-classified. The connector's wire behaviour is proven
// separately in FB_RobotConnector_Tests.
//
// Every test is a small scan-stepped sequencer: the sim's motion and the base's
// heartbeat are both TON-driven, so a loop of Cyclic() calls inside one scan
// advances no time at all. That mistake cost this suite two red tests once
// already; it is not repeated here.
FUNCTION_BLOCK FB_RobotCM_Tests EXTENDS TcUnit.FB_TestSuite
VAR
    _cmA : FB_RobotCM;  _rbA : FB_SimRobotConnector;  _sA : INT;  _nA : INT;
    _cmB : FB_RobotCM;  _rbB : FB_SimRobotConnector;  _sB : INT;  _nB : INT;
    _cmC : FB_RobotCM;  _rbC : FB_SimRobotConnector;  _sC : INT;  _nC : INT;
    _cmD : FB_RobotCM;  _rbD : FB_SimRobotConnector;  _sD : INT;  _nD : INT;
    _cmE : FB_RobotCM;  _rbE : FB_SimRobotConnector;  _sE : INT;  _nE : INT;
    _cmF : FB_RobotCM;  _rbF : FB_SimRobotConnector;  _sF : INT;  _nF : INT;
    _cmG : FB_RobotCM;  _rbG : FB_SimRobotConnector;  _sG : INT;  _nG : INT;
    _cmH : FB_RobotCM;  _rbH : FB_SimRobotConnector;  _sH : INT;  _nH : INT;
    _diag : ST_Diagnostic;   // C0185: cannot access .member on a property result
END_VAR

Command_on_a_down_link_faults_with_the_link_reason();
Motion_before_homing_is_refused();
Home_is_exempt_from_the_reference_check();
Speed_scale_outside_its_band_is_refused_before_motion();
Mode_that_does_not_permit_motion_is_refused();
Lost_permissive_holds_on_path_rather_than_faulting();
Completion_publishes_the_reached_position();
Protective_stop_aborts_with_its_own_reason();

METHOD PRIVATE Command_on_a_down_link_faults_with_the_link_reason
TEST('Command_on_a_down_link_faults_with_the_link_reason');
// Deliberately never Connect()ed: the connector stays down. A command must FAULT
// with the link reason rather than wait - a sequence blocked on a robot that
// never heard the command is the failure this rule exists to prevent (Annex D).
CASE _sA OF
    0:
        _cmA.Setup(Name := 'Test.RobotA', Robot := _rbA);
        _cmA.ParCfg.SpeedScaleMin := 1.0;
        _cmA.ParCfg.SpeedScaleMax := 100.0;
        _cmA.ParCmd.SpeedScale    := 50.0;
        _cmA.ParCmd.TargetId      := 5;
        _cmA.Command              := E_RobotCommand.MOVE_TO;
        _sA := 1;
    1:
        _cmA.Execute := TRUE;
        _cmA();
        _sA := 2;
    2:
        _cmA();
        IF _cmA.Error THEN
            _diag := _cmA.Status.Diagnostic;
            AssertEquals_DINT(Expected := E_Reason.LINK_TIMEOUT, Actual := _diag.ReasonCode,
                Message := 'a command on a down link faults with the link reason');
            AssertFalse(Condition := _cmA.Busy,
                Message := 'and does not sit BUSY waiting for a robot that never heard it');
            TEST_FINISHED();
        ELSE
            _nA := _nA + 1;
IF _nA > 2000 THEN
    AssertTrue(Condition := FALSE, Message := 'a command on a down link never faulted');
    TEST_FINISHED();
END_IF
        END_IF
END_CASE
END_METHOD

METHOD PRIVATE Motion_before_homing_is_refused
TEST('Motion_before_homing_is_refused');
// The heartbeat is TON-driven, so the link comes up over scans, not at once.
_rbB.Connect();
_rbB.Cyclic();

CASE _sB OF
    0:
        _cmB.Setup(Name := 'Test.RobotB', Robot := _rbB);
        _cmB.ParCfg.SpeedScaleMin := 1.0;
        _cmB.ParCfg.SpeedScaleMax := 100.0;
        _cmB.ParCfg.MoveTimeout   := T#2S;
        _cmB.ParCfg.HomeTimeout   := T#2S;
        _cmB.ParCfg.SpeedCeiling[E_RobotOpMode.AUTO_REMOTE] := 100.0;
        _cmB.ParCmd.SpeedScale    := 50.0;
        _cmB.ParCmd.TargetId      := 5;
        _cmB();
        IF _rbB.Linked THEN
            _rbB.PowerOn();          // powered but NEVER homed
            _sB := 1;
        END_IF
        _nB := _nB + 1;
IF _nB > 2000 THEN
    AssertTrue(Condition := FALSE, Message := 'the simulated link never came up');
    TEST_FINISHED();
END_IF
    1:
        _cmB.Command := E_RobotCommand.MOVE_TO;
        _cmB.Execute := TRUE;
        _cmB();
        _sB := 2;
    2:
        _cmB();
        IF _cmB.Error THEN
            // The specific cause, not the first check that happened to fail: an
            // unreferenced robot needs homing, and the operator is told exactly that.
            _diag := _cmB.Status.Diagnostic;
            AssertEquals_DINT(Expected := PL_ModuleReasons.ROBOT_NOT_REFERENCED,
                Actual := _diag.ReasonCode,
                Message := 'motion before homing is refused as unreferenced');
            AssertFalse(Condition := _rbB.MotionBusy,
                Message := 'and nothing was sent - the refusal is BEFORE motion (S5.6)');
            TEST_FINISHED();
        ELSE
            _nB := _nB + 1;
IF _nB > 2000 THEN
    AssertTrue(Condition := FALSE, Message := 'motion before homing was not refused');
    TEST_FINISHED();
END_IF
        END_IF
END_CASE
END_METHOD

METHOD PRIVATE Home_is_exempt_from_the_reference_check
TEST('Home_is_exempt_from_the_reference_check');
// The heartbeat is TON-driven, so the link comes up over scans, not at once.
_rbC.Connect();
_rbC.Cyclic();

// The ladder that refuses motion before homing must NOT refuse homing itself:
// homing is what ESTABLISHES the reference, so gating it on one would leave the
// robot permanently unhomeable - a deadlock the validation exists to prevent,
// not to create. This is the test that would have caught it.
CASE _sC OF
    0:
        _cmC.Setup(Name := 'Test.RobotC', Robot := _rbC);
        _cmC.ParCfg.SpeedScaleMin := 1.0;
        _cmC.ParCfg.SpeedScaleMax := 100.0;
        _cmC.ParCfg.MoveTimeout   := T#2S;
        _cmC.ParCfg.HomeTimeout   := T#2S;
        _cmC.ParCfg.SpeedCeiling[E_RobotOpMode.AUTO_REMOTE] := 100.0;
        _cmC.ParCmd.SpeedScale    := 50.0;
        _cmC();
        IF _rbC.Linked THEN
            _rbC.PowerOn();
            AssertFalse(Condition := _rbC.Referenced,
                Message := 'precondition: the robot starts unreferenced');
            _sC := 1;
        END_IF
        _nC := _nC + 1;
IF _nC > 2000 THEN
    AssertTrue(Condition := FALSE, Message := 'the simulated link never came up');
    TEST_FINISHED();
END_IF
    1:
        _cmC.Command := E_RobotCommand.HOME;
        _cmC.Execute := TRUE;
        _cmC();
        _sC := 2;
    2:
        _cmC();
        IF _cmC.Done THEN
            AssertTrue(Condition := _rbC.Referenced,
                Message := 'homing completes and establishes the reference');
            TEST_FINISHED();
        ELSIF _cmC.Error THEN
            _diag := _cmC.Status.Diagnostic;
            AssertEquals_DINT(Expected := 0, Actual := _diag.ReasonCode,
                Message := 'HOME must not be refused for being unreferenced');
            TEST_FINISHED();
        ELSE
            _nC := _nC + 1;
IF _nC > 2000 THEN
    AssertTrue(Condition := FALSE, Message := 'HOME neither completed nor faulted');
    TEST_FINISHED();
END_IF
        END_IF
END_CASE
END_METHOD

METHOD PRIVATE Speed_scale_outside_its_band_is_refused_before_motion
TEST('Speed_scale_outside_its_band_is_refused_before_motion');
// The heartbeat is TON-driven, so the link comes up over scans, not at once.
_rbD.Connect();
_rbD.Cyclic();

CASE _sD OF
    0:
        _cmD.Setup(Name := 'Test.RobotD', Robot := _rbD);
        _cmD.ParCfg.SpeedScaleMin := 10.0;
        _cmD.ParCfg.SpeedScaleMax := 80.0;
        _cmD.ParCfg.MoveTimeout   := T#2S;
        _cmD.ParCfg.HomeTimeout   := T#2S;
        _cmD.ParCfg.SpeedCeiling[E_RobotOpMode.AUTO_REMOTE] := 100.0;
        _cmD.ParCmd.SpeedScale    := 95.0;    // outside the configured band
        _cmD.ParCmd.TargetId      := 3;
        _cmD();
        IF _rbD.Linked THEN
            _rbD.PowerOn();
            _rbD.Home();
            _sD := 1;
        END_IF
        _nD := _nD + 1;
IF _nD > 2000 THEN
    AssertTrue(Condition := FALSE, Message := 'the simulated link never came up');
    TEST_FINISHED();
END_IF
    1:
        _cmD();
        IF _rbD.Referenced THEN
            _sD := 2;
        END_IF
        _nD := _nD + 1;
IF _nD > 2000 THEN
    AssertTrue(Condition := FALSE, Message := 'the simulated robot never homed');
    TEST_FINISHED();
END_IF
    2:
        _cmD.Command := E_RobotCommand.MOVE_TO;
        _cmD.Execute := TRUE;
        _cmD();
        _sD := 3;
    3:
        _cmD();
        IF _cmD.Error THEN
            // A malformed parameter is wrong regardless of mode or reference, so it
            // is checked FIRST and reported as itself.
            _diag := _cmD.Status.Diagnostic;
            AssertEquals_DINT(Expected := PL_ModuleReasons.ROBOT_PARAM_OOR,
                Actual := _diag.ReasonCode,
                Message := 'a speed scale outside the band is refused as out of range');
            AssertFalse(Condition := _rbD.MotionBusy,
                Message := 'and the robot never started moving');
            TEST_FINISHED();
        ELSE
            _nD := _nD + 1;
IF _nD > 2000 THEN
    AssertTrue(Condition := FALSE, Message := 'an out-of-band speed scale was not refused');
    TEST_FINISHED();
END_IF
        END_IF
END_CASE
END_METHOD

METHOD PRIVATE Mode_that_does_not_permit_motion_is_refused
TEST('Mode_that_does_not_permit_motion_is_refused');
// The heartbeat is TON-driven, so the link comes up over scans, not at once.
_rbE.Connect();
_rbE.Cyclic();

CASE _sE OF
    0:
        _cmE.Setup(Name := 'Test.RobotE', Robot := _rbE);
        _cmE.ParCfg.SpeedScaleMin := 1.0;
        _cmE.ParCfg.SpeedScaleMax := 100.0;
        _cmE.ParCfg.MoveTimeout   := T#2S;
        _cmE.ParCfg.HomeTimeout   := T#2S;
        _cmE.ParCfg.SpeedCeiling[E_RobotOpMode.AUTO_REMOTE]    := 100.0;
        _cmE.ParCfg.SpeedCeiling[E_RobotOpMode.MANUAL_REDUCED] := 25.0;
        _cmE.ParCmd.SpeedScale    := 50.0;
        _cmE.ParCmd.TargetId      := 3;
        _cmE();
        IF _rbE.Linked THEN
            _rbE.PowerOn();
            _rbE.Home();
            _sE := 1;
        END_IF
        _nE := _nE + 1;
IF _nE > 2000 THEN
    AssertTrue(Condition := FALSE, Message := 'the simulated link never came up');
    TEST_FINISHED();
END_IF
    1:
        _cmE();
        IF _rbE.Referenced THEN
            // The controller is put in a manual mode. Automatic motion commanded
            // from the PLC must not run in it, whatever the PLC would like.
            _rbE.RequestMode(Mode := E_RobotOpMode.MANUAL_REDUCED);
            _sE := 2;
        END_IF
        _nE := _nE + 1;
IF _nE > 2000 THEN
    AssertTrue(Condition := FALSE, Message := 'the simulated robot never homed');
    TEST_FINISHED();
END_IF
    2:
        _cmE.Command := E_RobotCommand.MOVE_TO;
        _cmE.Execute := TRUE;
        _cmE();
        _sE := 3;
    3:
        _cmE();
        IF _cmE.Error THEN
            _diag := _cmE.Status.Diagnostic;
            AssertEquals_DINT(Expected := PL_ModuleReasons.ROBOT_MODE_NOT_PERMITTED,
                Actual := _diag.ReasonCode,
                Message := 'the controllers REPORTED mode bounds what may run');
            AssertFalse(Condition := _rbE.MotionBusy,
                Message := 'and nothing was sent to the robot');
            TEST_FINISHED();
        ELSE
            _nE := _nE + 1;
IF _nE > 2000 THEN
    AssertTrue(Condition := FALSE, Message := 'a non-permitting mode did not refuse the move');
    TEST_FINISHED();
END_IF
        END_IF
END_CASE
END_METHOD

METHOD PRIVATE Lost_permissive_holds_on_path_rather_than_faulting
TEST('Lost_permissive_holds_on_path_rather_than_faulting');
// The heartbeat is TON-driven, so the link comes up over scans, not at once.
_rbF.Connect();
_rbF.Cyclic();

// S6.1, I.4b: losing a declared condition mid-move is EXPECTED - an operator
// releasing an enable is the designed way to stop a robot. It must HOLD, not
// fault: a fault would demand an acknowledgement for a normal act, and the
// alarm record would fill with events that were never faults.
CASE _sF OF
    0:
        _cmF.Setup(Name := 'Test.RobotF', Robot := _rbF);
        _cmF.DeclareCondition(Index := 1, DescriptionKey := 'std.interlock.areaSafe',
            Reason := E_Reason.INTERLOCK_DROPPED, Bypassable := FALSE);
        _cmF.SetCondition(Index := 1, Ok := TRUE);
        _cmF.ParCfg.SpeedScaleMin := 1.0;
        _cmF.ParCfg.SpeedScaleMax := 100.0;
        _cmF.ParCfg.MoveTimeout   := T#5S;
        _cmF.ParCfg.HomeTimeout   := T#5S;
        _cmF.ParCfg.SpeedCeiling[E_RobotOpMode.AUTO_REMOTE] := 100.0;
        _cmF.ParCmd.SpeedScale    := 50.0;
        _cmF.ParCmd.TargetId      := 4;
        _rbF.MoveTime := T#2S;                // long enough to interrupt mid-move
        _cmF();
        IF _rbF.Linked THEN
            _rbF.PowerOn();
            _rbF.Home();
            _sF := 1;
        END_IF
        _nF := _nF + 1;
IF _nF > 2000 THEN
    AssertTrue(Condition := FALSE, Message := 'the simulated link never came up');
    TEST_FINISHED();
END_IF
    1:
        _cmF.SetCondition(Index := 1, Ok := TRUE);
        _cmF();
        IF _rbF.Referenced THEN
            _sF := 2;
        END_IF
        _nF := _nF + 1;
IF _nF > 2000 THEN
    AssertTrue(Condition := FALSE, Message := 'the simulated robot never homed');
    TEST_FINISHED();
END_IF
    2:
        _cmF.SetCondition(Index := 1, Ok := TRUE);
        _cmF.Command := E_RobotCommand.MOVE_TO;
        _cmF.Execute := TRUE;
        _cmF();
        _sF := 3;
    3:
        _cmF.SetCondition(Index := 1, Ok := TRUE);
        _cmF();
        IF _rbF.MotionBusy THEN
            _sF := 4;                          // the arm is genuinely on its way
        END_IF
        _nF := _nF + 1;
IF _nF > 2000 THEN
    AssertTrue(Condition := FALSE, Message := 'the move never started');
    TEST_FINISHED();
END_IF
    4:
        _cmF.SetCondition(Index := 1, Ok := FALSE);   // the permissive drops
        _cmF();
        IF _cmF.Held THEN
            AssertFalse(Condition := _cmF.Error,
                Message := 'a lost permissive HOLDS - it is not a fault (S6.1)');
            AssertTrue(Condition := _cmF.Busy,
                Message := 'and the command is still BUSY, not terminated');
            _sF := 5;
        ELSE
            _nF := _nF + 1;
IF _nF > 2000 THEN
    AssertTrue(Condition := FALSE, Message := 'the lost permissive did not raise HELD');
    TEST_FINISHED();
END_IF
        END_IF
    5:
        // Level-based: the hold clears by itself the scan the condition returns,
        // with no per-type "clear the hold" code to forget.
        _cmF.SetCondition(Index := 1, Ok := TRUE);
        _cmF();
        IF NOT _cmF.Held THEN
            AssertFalse(Condition := _cmF.Error,
                Message := 'the restored permissive resumes rather than faulting');
            TEST_FINISHED();
        ELSE
            _nF := _nF + 1;
IF _nF > 2000 THEN
    AssertTrue(Condition := FALSE, Message := 'the hold never cleared after the condition returned');
    TEST_FINISHED();
END_IF
        END_IF
END_CASE
END_METHOD

METHOD PRIVATE Completion_publishes_the_reached_position
TEST('Completion_publishes_the_reached_position');
// The heartbeat is TON-driven, so the link comes up over scans, not at once.
_rbG.Connect();
_rbG.Cyclic();

CASE _sG OF
    0:
        _cmG.Setup(Name := 'Test.RobotG', Robot := _rbG);
        _cmG.ParCfg.SpeedScaleMin := 1.0;
        _cmG.ParCfg.SpeedScaleMax := 100.0;
        _cmG.ParCfg.MoveTimeout   := T#5S;
        _cmG.ParCfg.HomeTimeout   := T#5S;
        _cmG.ParCfg.SpeedCeiling[E_RobotOpMode.AUTO_REMOTE] := 100.0;
        _cmG.ParCmd.SpeedScale    := 50.0;
        _cmG.ParCmd.TargetId      := 7;
        _cmG();
        IF _rbG.Linked THEN
            _rbG.PowerOn();
            _rbG.Home();
            _sG := 1;
        END_IF
        _nG := _nG + 1;
IF _nG > 2000 THEN
    AssertTrue(Condition := FALSE, Message := 'the simulated link never came up');
    TEST_FINISHED();
END_IF
    1:
        _cmG();
        IF _rbG.Referenced THEN
            _sG := 2;
        END_IF
        _nG := _nG + 1;
IF _nG > 2000 THEN
    AssertTrue(Condition := FALSE, Message := 'the simulated robot never homed');
    TEST_FINISHED();
END_IF
    2:
        _cmG.Command := E_RobotCommand.MOVE_TO;
        _cmG.Execute := TRUE;
        _cmG();
        _sG := 3;
    3:
        _cmG();
        IF _cmG.Done THEN
            // OutCmd is what the COMMAND produced and stays latched until the next
            // one - distinct from OutImm, which is recomputed every scan (S3.12).
            AssertEquals_DWORD(Expected := 7, Actual := _cmG.OutCmd.ReachedId,
                Message := 'completion publishes the position actually reached');
            AssertTrue(Condition := _cmG.OutImm.Linked,
                Message := 'and the live facts mirror the connector');
            AssertFalse(Condition := _cmG.OutImm.MotionBusy,
                Message := 'with motion finished');
            TEST_FINISHED();
        ELSIF _cmG.Error THEN
            _diag := _cmG.Status.Diagnostic;
            AssertEquals_DINT(Expected := 0, Actual := _diag.ReasonCode,
                Message := 'the move should have completed, not faulted');
            TEST_FINISHED();
        ELSE
            _nG := _nG + 1;
IF _nG > 2000 THEN
    AssertTrue(Condition := FALSE, Message := 'the move neither completed nor faulted');
    TEST_FINISHED();
END_IF
        END_IF
END_CASE
END_METHOD

METHOD PRIVATE Protective_stop_aborts_with_its_own_reason
TEST('Protective_stop_aborts_with_its_own_reason');
// The heartbeat is TON-driven, so the link comes up over scans, not at once.
_rbH.Connect();
_rbH.Cyclic();

// I.4a(c): the robot's crash device is NOT a S9 safety function, and must never
// be recorded as one. A process event filed as a safety event corrupts exactly
// the record a safety review reads.
CASE _sH OF
    0:
        _cmH.Setup(Name := 'Test.RobotH', Robot := _rbH);
        _cmH.ParCfg.SpeedScaleMin := 1.0;
        _cmH.ParCfg.SpeedScaleMax := 100.0;
        _cmH.ParCfg.MoveTimeout   := T#5S;
        _cmH.ParCfg.HomeTimeout   := T#5S;
        _cmH.ParCfg.SpeedCeiling[E_RobotOpMode.AUTO_REMOTE] := 100.0;
        _cmH.ParCmd.SpeedScale    := 50.0;
        _cmH.ParCmd.TargetId      := 6;
        _rbH.MoveTime := T#2S;
        _cmH();
        IF _rbH.Linked THEN
            _rbH.PowerOn();
            _rbH.Home();
            _sH := 1;
        END_IF
        _nH := _nH + 1;
IF _nH > 2000 THEN
    AssertTrue(Condition := FALSE, Message := 'the simulated link never came up');
    TEST_FINISHED();
END_IF
    1:
        _cmH();
        IF _rbH.Referenced THEN
            _sH := 2;
        END_IF
        _nH := _nH + 1;
IF _nH > 2000 THEN
    AssertTrue(Condition := FALSE, Message := 'the simulated robot never homed');
    TEST_FINISHED();
END_IF
    2:
        _cmH.Command := E_RobotCommand.MOVE_TO;
        _cmH.Execute := TRUE;
        _cmH();
        _sH := 3;
    3:
        _cmH();
        IF _rbH.MotionBusy THEN
            _rbH.Inject := E_RobotSimFault.PROTECTIVE_STOP;   // the crash device trips
            _sH := 4;
        END_IF
        _nH := _nH + 1;
IF _nH > 2000 THEN
    AssertTrue(Condition := FALSE, Message := 'the move never started');
    TEST_FINISHED();
END_IF
    4:
        _cmH();
        IF _cmH.Error THEN
            _diag := _cmH.Status.Diagnostic;
            AssertEquals_DINT(Expected := PL_ModuleReasons.ROBOT_PROTECTIVE_STOP,
                Actual := _diag.ReasonCode,
                Message := 'a protective stop faults with its OWN reason, not a safety one');
            AssertTrue(Condition := _cmH.OutImm.ProtectiveStop,
                Message := 'and the condition is published while it stands');
            TEST_FINISHED();
        ELSE
            _nH := _nH + 1;
IF _nH > 2000 THEN
    AssertTrue(Condition := FALSE, Message := 'the protective stop did not fault the command');
    TEST_FINISHED();
END_IF
        END_IF
END_CASE
END_METHOD

END_FUNCTION_BLOCK

// ---- Fraktal_Tests/FB_AxisJog_Tests.TcPOU
// Core §9 / §7.6.1 — jogging an axis by hand under a safety-rated enabling
// device, and the derivation that decides whether one is permitting.
//
// The derivation tests matter more than they look: every one of them is a way a
// cell could end up jogging with its guards open when it should not. They are
// written as the fail-closed cases first, because that is the direction in which
// being wrong is dangerous.
FUNCTION_BLOCK FB_AxisJog_Tests EXTENDS TcUnit.FB_TestSuite
VAR
    _sfy  : ST_SafetyStatus;
    _en   : ST_ManualEnableStatus;
    _axA  : FB_AxisCM;   _refA : AXIS_REF;   _sA : INT;   _nA : INT;
    _axB  : FB_AxisCM;   _refB : AXIS_REF;   _sB : INT;   _nB : INT;
    _axC  : FB_AxisCM;   _refC : AXIS_REF;
    _w1, _w2, _w3, _w4, _w5, _w6, _w7 : BOOL;
END_VAR

No_enabling_device_mirrored_means_never_enabled();
A_released_enabling_device_does_not_permit();
A_held_enabling_device_permits_and_names_itself();
A_safety_fault_withdraws_the_permission();
Jog_is_refused_without_a_held_enabling_device();
Jog_stops_when_the_request_stops_arriving();
Capture_stores_the_modules_own_live_value();
Capture_is_refused_for_a_key_that_offers_none();

// Build a safety facet carrying one enabling device in a given state.
METHOD PRIVATE _M_Enable
VAR_INPUT
    Permitting : BOOL;
    Faulted    : BOOL;
END_VAR
_sfy.Present := TRUE;
_sfy.FaultActive := Faulted;
_sfy.Devices[1].Present         := TRUE;
_sfy.Devices[1].Name            := 'TeachEnable01';
_sfy.Devices[1].Kind            := E_SafetyDeviceKind.ENABLE_SWITCH;
_sfy.Devices[1].FieldbusHealthy := TRUE;
// Permitting is the POSITIVE state, exactly as for an E-stop that is not pressed.
_sfy.Devices[1].Ready           := Permitting;
_sfy.Devices[1].DemandActive    := NOT Permitting;
_sfy.Devices[1].SafeStateActive := NOT Permitting;
_sfy.Devices[1].FaultActive     := FALSE;
_sfy.Devices[1].State           := SEL(Permitting, E_SafetyState.DEMAND, E_SafetyState.READY);
END_METHOD

METHOD PRIVATE No_enabling_device_mirrored_means_never_enabled
TEST('No_enabling_device_mirrored_means_never_enabled');
IF NOT _w1 THEN
    // A cell that never wired an enabling device must not be able to jog with the
    // guards open BY OMISSION. Absence is the commonest way this goes wrong, so
    // it is the first case.
    MEMSET(ADR(_sfy), 0, SIZEOF(_sfy));
    _en := F_ManualEnable(Safety := _sfy);
    AssertFalse(Condition := _en.Present, Message := 'no device is reported as present');
    AssertFalse(Condition := _en.Held,    Message := 'and nothing is permitting');

    // A safety facet that exists but carries only OTHER kinds is the same answer.
    _sfy.Present := TRUE;
    _sfy.Devices[1].Present := TRUE;
    _sfy.Devices[1].Kind    := E_SafetyDeviceKind.GUARD_DOOR;
    _sfy.Devices[1].Ready   := TRUE;
    _en := F_ManualEnable(Safety := _sfy);
    AssertFalse(Condition := _en.Held,
        Message := 'a closed guard is not an enabling device');
    _w1 := TRUE;
END_IF
TEST_FINISHED();
END_METHOD

METHOD PRIVATE A_released_enabling_device_does_not_permit
TEST('A_released_enabling_device_does_not_permit');
IF NOT _w2 THEN
    // Released AND panic-squeezed are the same answer here, which is the whole
    // reason the device has three positions rather than two: both non-middle
    // positions demand the safe state.
    _M_Enable(Permitting := FALSE, Faulted := FALSE);
    _en := F_ManualEnable(Safety := _sfy);
    AssertTrue(Condition := _en.Present,
        Message := 'the device is mirrored');
    AssertFalse(Condition := _en.Held,
        Message := 'but it is not permitting, so nothing may move');
    _w2 := TRUE;
END_IF
TEST_FINISHED();
END_METHOD

METHOD PRIVATE A_held_enabling_device_permits_and_names_itself
TEST('A_held_enabling_device_permits_and_names_itself');
IF NOT _w3 THEN
    _M_Enable(Permitting := TRUE, Faulted := FALSE);
    _en := F_ManualEnable(Safety := _sfy);
    AssertTrue(Condition := _en.Held,
        Message := 'a held enabling device permits manual motion');
    // Named so a release report can say WHICH device, rather than "not released".
    AssertEquals_STRING(Expected := 'TeachEnable01', Actual := _en.DeviceName,
        Message := 'and names itself for the release report (S7.6.0)');
    _w3 := TRUE;
END_IF
TEST_FINISHED();
END_METHOD

METHOD PRIVATE A_safety_fault_withdraws_the_permission
TEST('A_safety_fault_withdraws_the_permission');
IF NOT _w4 THEN
    // The device still reads as held, but the safety system is reporting a fault.
    // A safety system that is not healthy is not one to take permission from.
    _M_Enable(Permitting := TRUE, Faulted := TRUE);
    _en := F_ManualEnable(Safety := _sfy);
    AssertFalse(Condition := _en.Held,
        Message := 'a faulted safety facet grants nothing, however the switch reads');

    // Same for the device's own fieldbus: a stale mirror is not a permission.
    _M_Enable(Permitting := TRUE, Faulted := FALSE);
    _sfy.Devices[1].FieldbusHealthy := FALSE;
    _en := F_ManualEnable(Safety := _sfy);
    AssertFalse(Condition := _en.Held,
        Message := 'and neither does an unhealthy safety fieldbus');
    _w4 := TRUE;
END_IF
TEST_FINISHED();
END_METHOD

METHOD PRIVATE Jog_is_refused_without_a_held_enabling_device
TEST('Jog_is_refused_without_a_held_enabling_device');
IF NOT _w5 THEN
    _axA.Setup(Name := 'Test.AxisA', AxisRef := _refA, Recipe := 0);
    _axA.DeclareCondition(Index := 1, DescriptionKey := 'std.interlock.areaSafe',
        Reason := E_Reason.INTERLOCK_DROPPED, Bypassable := FALSE);
    _axA.SetCondition(Index := 1, Ok := TRUE);

    // Not permitting -> the request is refused at the door, with its reason.
    _M_Enable(Permitting := FALSE, Faulted := FALSE);
    _en := F_ManualEnable(Safety := _sfy);
    AssertFalse(Condition := _axA.RequestHeldCommand(
            Value := TO_DINT(E_AxisCommand.JOG_POS), Enable := _en),
        Message := 'jog is refused when no enabling device is permitting');
    _axA();
    AssertFalse(Condition := _axA.OutImm.Jogging,
        Message := 'and the axis is not jogging');
    AssertEquals_DINT(Expected := PL_ModuleReasons.AXIS_JOG_NOT_ENABLED,
        Actual := _axA.OutImm.JogStopReason,
        Message := 'the operator is told why, not left guessing (O3)');

    // An unknown held value is refused too, and leaves no direction behind (S5.6).
    _M_Enable(Permitting := TRUE, Faulted := FALSE);
    _en := F_ManualEnable(Safety := _sfy);
    AssertFalse(Condition := _axA.RequestHeldCommand(Value := 9999, Enable := _en),
        Message := 'an unknown held command is refused');
    _axA();
    AssertFalse(Condition := _axA.OutImm.Jogging,
        Message := 'and starts no motion');
    _w5 := TRUE;
END_IF
TEST_FINISHED();
END_METHOD

METHOD PRIVATE Jog_stops_when_the_request_stops_arriving
TEST('Jog_stops_when_the_request_stops_arriving');
// O10, and the reason this whole surface is level-driven: a held jog delivered
// over a network must stop when the asking stops - whether the operator let go
// or the transport died. Runs ACROSS SCANS because the deadline is a TON.
CASE _sB OF
    0:
        _axB.Setup(Name := 'Test.AxisB', AxisRef := _refB, Recipe := 0);
        _axB.DeclareCondition(Index := 1, DescriptionKey := 'std.interlock.areaSafe',
            Reason := E_Reason.INTERLOCK_DROPPED, Bypassable := FALSE);
        _axB.ParCfg.JogTimeout := T#100MS;
        _sB := 1;
    1:
        // Ask every scan, as a held control does, with everything permitting.
        _axB.SetCondition(Index := 1, Ok := TRUE);
        _M_Enable(Permitting := TRUE, Faulted := FALSE);
        _en := F_ManualEnable(Safety := _sfy);
        _axB.RequestHeldCommand(Value := TO_DINT(E_AxisCommand.JOG_POS), Enable := _en);
        _axB();
        IF _axB.OutImm.Jogging THEN
            _sB := 2;
        END_IF
        _nB := _nB + 1;
        IF _nB > 2000 THEN
            AssertTrue(Condition := FALSE, Message := 'the jog never started');
            TEST_FINISHED();
        END_IF
    2:
        // Now stop asking. Nothing else changes: the interlock still holds and the
        // enabling device is still held. Only the asking stopped.
        _axB.SetCondition(Index := 1, Ok := TRUE);
        _axB();
        IF NOT _axB.OutImm.Jogging THEN
            AssertEquals_DINT(Expected := PL_ModuleReasons.AXIS_JOG_RELEASED,
                Actual := _axB.OutImm.JogStopReason,
                Message := 'and says the request stopped arriving');
            TEST_FINISHED();
        END_IF
        _nB := _nB + 1;
        IF _nB > 4000 THEN
            AssertTrue(Condition := FALSE,
                Message := 'the axis kept jogging after the requests stopped');
            TEST_FINISHED();
        END_IF
END_CASE
END_METHOD

METHOD PRIVATE Capture_stores_the_modules_own_live_value
TEST('Capture_stores_the_modules_own_live_value');
IF NOT _w6 THEN
    // §3.8c: the point of jogging is to keep where you got to. The capture writes
    // the module's OWN published ActPos into its OWN registered field - it does
    // not accept a number from the client, which is what makes it a capture.
    _axC.Setup(Name := 'Test.AxisC', AxisRef := _refC, Recipe := 0);
    _axC();
    AssertTrue(Condition := _axC.M_ApplyCapture(Scope := 'Test.AxisC',
            WriteKey := 'axis.taughtPosition', Revision := 1, RootReady := TRUE),
        Message := 'the capture is accepted by the field that registered it');
    _axC();
    AssertEquals_LREAL(Expected := _axC.OutImm.ActPos,
        Actual := _axC.OutImm.TaughtPosition, Delta := 0.0001,
        Message := 'and the stored value IS the live one, not a client-supplied number');
    _w6 := TRUE;
END_IF
TEST_FINISHED();
END_METHOD

METHOD PRIVATE Capture_is_refused_for_a_key_that_offers_none
TEST('Capture_is_refused_for_a_key_that_offers_none');
IF NOT _w7 THEN
    // An unregistered key stores nothing. Falling back to a default here would let
    // an unoffered capture quietly write a zero over a taught position (§5.6).
    AssertFalse(Condition := _axC.M_ApplyCapture(Scope := 'Test.AxisC',
            WriteKey := 'axis.notAThing', Revision := 1, RootReady := TRUE),
        Message := 'an unknown key is refused');
    // A stale revision is refused on the capture path too, because the capture
    // rejoins the ordinary write path rather than going around it (§3.8c).
    AssertFalse(Condition := _axC.M_ApplyCapture(Scope := 'Test.AxisC',
            WriteKey := 'axis.taughtPosition', Revision := 99, RootReady := TRUE),
        Message := 'and so is a stale revision - same validation as a typed write');
    _w7 := TRUE;
END_IF
TEST_FINISHED();
END_METHOD

END_FUNCTION_BLOCK

// ---- Fraktal_Tests/FB_Separator_Tests.TcPOU
// Annex A separator/stopper. T1/T4 are proven once in FB_Base_Tests for every
// inheriting type and are deliberately NOT repeated here (Core S5.7).
//
// The first test is the one that matters most: this type declares NO interlocks
// of its own (S7.2.1), so the suite proves both halves of that contract - nothing
// gates a station that declares nothing, and a condition the application declares
// is fail-closed until the application drives it.
FUNCTION_BLOCK FB_Separator_Tests EXTENDS TcUnit.FB_TestSuite
VAR
    _hal : ST_SeparatorHal;
    _sep : FB_SeparatorCM;
    _halT3 : ST_SeparatorHal;
    _sepT3 : FB_SeparatorCM;
    _halSep : ST_SeparatorHal;
    _sepSep : FB_SeparatorCM;
    _halNo : ST_SeparatorHal;
    _sepNo : FB_SeparatorCM;
    _halOc : ST_SeparatorHal;
    _sepOc : FB_SeparatorCM;
    _halBad : ST_SeparatorHal;
    _sepBad : FB_SeparatorCM;
    _i : INT;
    _w1, _w2, _w3, _w4, _w5, _w6 : BOOL;
END_VAR

Library_declares_no_interlocks_and_application_conditions_are_fail_closed();
Interlock_withholds_the_valve_and_holds_rather_than_faults();
Separate_releases_one_carrier_and_completes();
No_carrier_at_the_separator_faults_10001();
Open_close_confirms_feedback_only_when_configured();
Unsupported_command_is_rejected();

METHOD Library_declares_no_interlocks_and_application_conditions_are_fail_closed
TEST('Library_declares_no_interlocks_and_application_conditions_are_fail_closed');
IF NOT _w1 THEN
    _sep.Setup(Name := 'Sep1', HalRef := _hal, Recipe := 0);
    _sep();
    // S7.2.1: a reusable type publishes no condition it cannot derive. A station
    // that declares nothing is therefore not gated by anything.
    AssertTrue(Condition := _sep.Intlk.AllOk,
        Message := 'a library type that declares no interlock does not gate the station');
    AssertTrue(Condition := _sep.DeclareCondition(Index := 1,
            DescriptionKey := 'std.interlock.areaSafe',
            Reason := E_Reason.INTERLOCK_DROPPED, Bypassable := FALSE),
        Message := 'the application may claim any index');
    _sep();
    // Declaring states an intent to gate, so the fail-closed default holds until
    // the application actually drives it.
    AssertFalse(Condition := _sep.Intlk.AllOk,
        Message := 'a declared but undriven condition is fail-closed');
    AssertTrue(Condition := _sep.SetCondition(Index := 1, Ok := TRUE),
        Message := 'the application drives its own condition');
    _sep();
    AssertTrue(Condition := _sep.Intlk.AllOk,
        Message := 'and the gate clears once it is satisfied');
    AssertFalse(Condition := _sep.DeclareCondition(Index := 0,
            DescriptionKey := 'std.interlock.areaSafe',
            Reason := E_Reason.INTERLOCK_DROPPED, Bypassable := FALSE),
        Message := 'an out-of-range index is refused, not silently ignored');
    _w1 := TRUE;
END_IF
TEST_FINISHED();
END_METHOD

METHOD Interlock_withholds_the_valve_and_holds_rather_than_faults
TEST('Interlock_withholds_the_valve_and_holds_rather_than_faults');
IF NOT _w2 THEN
    _sepT3.Setup(Name := 'SepT3', HalRef := _halT3, Recipe := 0);
    _sepT3.DeclareCondition(Index := 1, DescriptionKey := 'std.interlock.areaSafe',
        Reason := E_Reason.INTERLOCK_DROPPED, Bypassable := FALSE);
    _sepT3.SetCondition(Index := 1, Ok := FALSE);
    _halT3.CarrierAt := TRUE;
    _sepT3.Command := E_SeparatorCommand.SEPARATE;
    _sepT3.Execute := TRUE;
    FOR _i := 1 TO 5 DO
        _sepT3();
    END_FOR
    // T3: the interlock withholds the output, and does so as a HELD wait rather
    // than a fault - losing a condition mid-action is expected, not a defect.
    AssertFalse(Condition := _halT3.ValveOpen,
        Message := 'the valve is withheld while the condition is unsatisfied');
    AssertTrue(Condition := _sepT3.Held, Message := 'and the module reports HELD');
    AssertFalse(Condition := _sepT3.Error, Message := 'not an error');
    AssertEquals_STRING(Expected := 'SepT3', Actual := _sepT3.Status.Diagnostic.SourcePath,
        Message := 'the owning module sets the diagnostic source path');
    _w2 := TRUE;
END_IF
TEST_FINISHED();
END_METHOD

METHOD Separate_releases_one_carrier_and_completes
TEST('Separate_releases_one_carrier_and_completes');
IF NOT _w3 THEN
    _sepSep.Setup(Name := 'SepOk', HalRef := _halSep, Recipe := 0);
    _sepSep.ParCfg.CheckAfter := FALSE;          // stopper variant: no downstream sensor
    _halSep.CarrierAt := TRUE;
    _sepSep.Command := E_SeparatorCommand.SEPARATE;
    _sepSep.Execute := TRUE;
    _sepSep(); _sepSep();
    AssertTrue(Condition := _halSep.ValveOpen, Message := 'opening drives the valve');
    _halSep.CarrierAt := FALSE;                  // the carrier leaves the separator
    _sepSep(); _sepSep(); _sepSep();
    AssertTrue(Condition := _sepSep.Done, Message := 'the command completes');
    AssertTrue(Condition := _sepSep.OutCmd.SeparateOk, Message := 'and reports the release');
    AssertFalse(Condition := _halSep.ValveOpen, Message := 'with the valve closed again');
    _w3 := TRUE;
END_IF
TEST_FINISHED();
END_METHOD

METHOD No_carrier_at_the_separator_faults_10001
TEST('No_carrier_at_the_separator_faults_10001');
IF NOT _w4 THEN
    _sepNo.Setup(Name := 'SepNo', HalRef := _halNo, Recipe := 0);
    // T#0S is the deterministic-timeout idiom used by the sibling suites: a TON
    // with PT := T#0S expires on the call that starts it, so the expiry does not
    // depend on task time elapsing. Calling the FB N times inside one test scan
    // does NOT advance a TON, which is why a small non-zero PT never fires here.
    _sepNo.ParCfg.MaxOpenTime := T#0S;
    _halNo.CarrierAt := FALSE;                   // nothing ever arrives
    _sepNo.Command := E_SeparatorCommand.SEPARATE;
    _sepNo.Execute := TRUE;
    _sepNo(); _sepNo(); _sepNo();
    // T2: the first-out reason is the specific one, not a generic timeout.
    AssertTrue(Condition := _sepNo.Error, Message := 'the command faults');
    AssertEquals_DWORD(Expected := TO_DWORD(PL_ModuleReasons.SEP_NO_CARRIER_AT),
        Actual := _sepNo.ErrorID,
        Message := 'with SEP_NO_CARRIER_AT, not a generic timeout');
    AssertEquals_STRING(Expected := 'SepNo', Actual := _sepNo.Status.Diagnostic.SourcePath,
        Message := 'and the module as its source path');
    AssertFalse(Condition := _halNo.ValveOpen, Message := 'the valve is dropped on fault');
    _w4 := TRUE;
END_IF
TEST_FINISHED();
END_METHOD

METHOD Open_close_confirms_feedback_only_when_configured
TEST('Open_close_confirms_feedback_only_when_configured');
IF NOT _w5 THEN
    _sepOc.Setup(Name := 'SepOc', HalRef := _halOc, Recipe := 0);
    _sepOc.ParCfg.UsesOpenFb := FALSE;           // no feedback wired at this station
    _sepOc.ParCmd.OpenStopper := TRUE;
    _sepOc.Command := E_SeparatorCommand.OPEN_CLOSE;
    _sepOc.Execute := TRUE;
    _sepOc(); _sepOc();
    AssertTrue(Condition := _halOc.ValveOpen, Message := 'the stopper opens');
    AssertTrue(Condition := _sepOc.Done,
        Message := 'and completes without feedback when none is configured');
    _sepOc.Execute := FALSE;
    _sepOc();
    _sepOc.ParCmd.OpenStopper := FALSE;
    _sepOc.Execute := TRUE;
    _sepOc(); _sepOc();
    AssertFalse(Condition := _halOc.ValveOpen, Message := 'closing is immediate');
    AssertTrue(Condition := _sepOc.Done, Message := 'and completes');
    _w5 := TRUE;
END_IF
TEST_FINISHED();
END_METHOD

METHOD Unsupported_command_is_rejected
TEST('Unsupported_command_is_rejected');
IF NOT _w6 THEN
    _sepBad.Setup(Name := 'SepBad', HalRef := _halBad, Recipe := 0);
    _sepBad.Command := E_SeparatorCommand.NONE;   // never a valid request (S5.6)
    _sepBad.Execute := TRUE;
    _sepBad(); _sepBad();
    AssertTrue(Condition := _sepBad.Error, Message := 'an unset command is refused');
    AssertEquals_DWORD(Expected := TO_DWORD(E_Reason.UNSUPPORTED_COMMAND),
        Actual := _sepBad.ErrorID, Message := 'with UNSUPPORTED_COMMAND');
    _w6 := TRUE;
END_IF
TEST_FINISHED();
END_METHOD

END_FUNCTION_BLOCK

// ---- Fraktal_Tests/FB_Engineering_Tests.TcPOU
// Core §7.5 under test: the gate register is write-once and build-driven, the
// standing §7.5.2 annunciation is LOW/SYSTEM/AUTO_RESET, no operator action
// closes it, and §10.5.1 forcing is refused unless the register arms it.
//
// The assertions about OUTPUT_FORCING are written against
// PL_FraktalEngineering.OUTPUT_FORCING rather than against TRUE or FALSE, so the
// suite is green in BOTH images and proves the two are actually coupled - a test
// hard-coded to the production value would pass while the commissioning build
// silently armed nothing.
FUNCTION_BLOCK FB_Engineering_Tests EXTENDS TcUnit.FB_TestSuite
VAR
    _mode : FB_EngineeringMode;
    _overflow : FB_EngineeringMode;
    _u : FB_ProbeUnit;
    _gateMode : FB_EngineeringMode;
    _i : INT;
    _slot : INT;
    _second : INT;
    _w1, _w2, _w3, _w4 : BOOL;
END_VAR

Inactive_gate_is_not_registered_and_declaring_is_idempotent();
Register_overflow_is_reported_not_silent();
Forcing_is_armed_only_by_the_build_constant();
Active_gate_annunciates_low_system_and_no_reset_closes_it();

METHOD Inactive_gate_is_not_registered_and_declaring_is_idempotent
TEST('Inactive_gate_is_not_registered_and_declaring_is_idempotent');
IF NOT _w1 THEN
    // §7.5.1: an inactive gate registers NOTHING - that is what makes a
    // production station's register empty and its gated surfaces invisible
    // rather than merely disabled.
    AssertEquals_INT(Expected := 0,
        Actual := _mode.M_Declare(Name := 'USE_SIMULATION',
            DescriptionKey := 'std.engineering.simulation', Active := FALSE),
        Message := 'an inactive gate is not registered');
    AssertEquals_INT(Expected := 0, Actual := _mode.Count,
        Message := 'so the register stays empty');
    _slot := _mode.M_Declare(Name := 'USE_SIMULATION',
        DescriptionKey := 'std.engineering.simulation', Active := TRUE);
    AssertTrue(Condition := _slot > 0, Message := 'an active gate is registered');
    AssertEquals_STRING(Expected := 'std.engineering.simulation',
        Actual := _mode.Gates[_slot].DescriptionKey,
        Message := 'with the key the standing annunciation will carry');
    // Re-declaring keeps the slot: two callers naming one departure must not
    // produce two standing annunciations for it.
    _second := _mode.M_Declare(Name := 'USE_SIMULATION',
        DescriptionKey := 'std.engineering.simulation', Active := TRUE);
    AssertEquals_INT(Expected := _slot, Actual := _second,
        Message := 'declaring the same gate again keeps its slot');
    AssertEquals_INT(Expected := 1, Actual := _mode.Count,
        Message := 'and does not grow the register');
    AssertFalse(Condition := _mode.Truncated, Message := 'nothing was dropped');
    _w1 := TRUE;
END_IF
TEST_FINISHED();
END_METHOD

METHOD Register_overflow_is_reported_not_silent
VAR
    gateName : STRING(80);
END_VAR
TEST('Register_overflow_is_reported_not_silent');
IF NOT _w2 THEN
    FOR _i := 1 TO PL_Fraktal.MAX_ENGINEERING_GATES + 1 DO
        gateName := CONCAT('GATE_', INT_TO_STRING(_i));
        _overflow.M_Declare(Name := gateName,
            DescriptionKey := 'std.engineering.simulation', Active := TRUE);
    END_FOR
    AssertEquals_INT(Expected := PL_Fraktal.MAX_ENGINEERING_GATES,
        Actual := _overflow.Count, Message := 'the table is bounded (O10)');
    // A gate that overflowed the table would otherwise be a departure nobody is
    // told about - the exact failure §7.5.2 exists to prevent (§5.6).
    AssertTrue(Condition := _overflow.Truncated,
        Message := 'and says so instead of dropping a gate silently');
    _w2 := TRUE;
END_IF
TEST_FINISHED();
END_METHOD

METHOD Forcing_is_armed_only_by_the_build_constant
TEST('Forcing_is_armed_only_by_the_build_constant');
IF NOT _w3 THEN
    // Before anything wires the register, forcing is refused: an unwired Unit is
    // a production Unit (§10.5.1 rule 1, fail closed).
    AssertFalse(Condition := _u.M_ForcePermitted(),
        Message := 'no register wired, so no forcing');
    AssertFalse(Condition := _u.ForceChannel(ChannelPath := 'Test.IO.X',
        Force := TRUE, BoolText := 'true', AnalogText := '0'),
        Message := 'and the request is refused before any resolver runs');
    _u.SetEngineeringMode(Mode := _gateMode);
    AssertTrue(Condition := (_gateMode.ForcingActive = PL_FraktalEngineering.OUTPUT_FORCING),
        Message := 'wiring the register arms forcing iff the build constant says so');
    AssertTrue(Condition := ((_gateMode.Count > 0) = PL_FraktalEngineering.OUTPUT_FORCING),
        Message := 'and an armed force surface always brings its gate with it');
    _w3 := TRUE;
END_IF
TEST_FINISHED();
END_METHOD

METHOD Active_gate_annunciates_low_system_and_no_reset_closes_it
TEST('Active_gate_annunciates_low_system_and_no_reset_closes_it');
IF NOT _w4 THEN
    AssertTrue(Condition := _u.Setup(Name := 'Test.GateUnit'), Message := 'unit sets up');
    _u.SetEngineeringMode(Mode := _gateMode);
    _gateMode.M_Declare(Name := 'USE_SIMULATION',
        DescriptionKey := 'std.engineering.simulation', Active := TRUE);
    _u();
    _slot := _u.AlarmLog.FindActiveSlot(SourcePath := 'Test.GateUnit',
        Description := 'std.engineering.simulation');
    AssertTrue(Condition := _slot > 0, Message := 'the gate is annunciated');
    AssertEquals_DINT(Expected := TO_DINT(E_Severity.LOW),
        Actual := TO_DINT(_u.AlarmLog.Active[_slot].Severity),
        Message := 'at the LOWEST priority (§8.1)');
    AssertEquals_DINT(Expected := TO_DINT(E_Category.SYSTEM),
        Actual := TO_DINT(_u.AlarmLog.Active[_slot].Category),
        Message := 'in the SYSTEM class: this is about the build, not the process');
    AssertEquals_DINT(Expected := TO_DINT(E_ResetClass.AUTO_RESET),
        Actual := TO_DINT(_u.AlarmLog.Active[_slot].ResetClass),
        Message := 'AUTO_RESET, so it never blocks the commissioning it serves');
    AssertFalse(Condition := _u.AlarmLog.Blocking,
        Message := 'and Start stays available');
    // The whole point: no operator action closes this. OperatorReset reaches
    // only MANUAL_RESET events, and the rationalization record is not shelvable.
    _u.AlarmLog.OperatorReset();
    _u();
    AssertTrue(Condition := _u.AlarmLog.FindActiveSlot(SourcePath := 'Test.GateUnit',
        Description := 'std.engineering.simulation') > 0,
        Message := 'an operator reset does not clear it');
    AssertFalse(Condition := _u.AlarmLog.Shelve(Slot := _slot, DurationS := 60),
        Message := 'and shelving cannot silence it either');
    // It is raised ONCE per gate, however long the station runs.
    _u();
    _u();
    AssertEquals_INT(Expected := _gateMode.Count, Actual := _u.AlarmLog.NActive,
        Message := 'one standing event per REGISTERED gate, not one per scan');
    _w4 := TRUE;
END_IF
TEST_FINISHED();
END_METHOD

END_FUNCTION_BLOCK

// ---- Fraktal_Tests/FB_ConfigDurability_Tests.TcPOU
// Core §3.8b under test, the half that is about TIME rather than content:
//
//   * a retained image is restored, or the module runs on declared defaults -
//     and the difference between "never written" and "written by a build that
//     laid it out differently" is the difference between silence and an alarm;
//   * an accepted write is LIVE, and stays PUBLISHED AS NOT DURABLE until the
//     store says otherwise, within a window the deployment declares;
//   * what a lost image COSTS is the deployment's declaration, not the module's:
//     the same loss either annunciates and runs, or refuses START_STOP until an
//     ENGINEER acknowledges it.
//
// The fixture is the same FB_ProbeConfigUnit/FB_ProbeConfigCM pair the §3.10.2
// write suite uses, on purpose: neither probe contains one line of persistence
// code, so if these pass, a station gets all of it for free (§1.1 O1).
FUNCTION_BLOCK FB_ConfigDurability_Tests EXTENDS TcUnit.FB_TestSuite
VAR
    _u        : FB_ProbeConfigUnit;
    _init     : BOOL;
    _store    : FB_LocalConfigStore;
    _persist  : FB_ProbeConfigPersistence;
    _users    : FB_LocalAccessProvider;
    _report   : ST_ReleaseReport;
    _version  : UINT;                 // a stand-in retained StationCfg image
    _path     : STRING(80);
    _expected : UINT;
    _found    : UINT;
    _taken    : BOOL;
    _released : BOOL;
    _i        : INT;
    // The window test is the one test here that must span scans (TIME() does not
    // advance inside one), so the other seven run exactly once: re-run each scan,
    // their writes would re-arm the very window being measured.
    _firstPass : BOOL;
    _winArmed  : BOOL;
    _winScans  : INT;
END_VAR

IF NOT _firstPass THEN
    _firstPass := TRUE;
    First_boot_initializes_silently();
    A_matching_version_restores_and_reports_nothing();
    An_unrecognized_version_is_reported_once_with_its_owner();
    The_root_annunciates_a_loss_without_blocking_on_its_own();
    Blocking_policy_refuses_start_until_an_engineer_acknowledges();
    An_accepted_write_is_pending_until_the_store_completes();
    A_store_that_refuses_publishes_PersistFailed();
END_IF
An_elapsed_window_publishes_PersistFailed();

// One-time wiring, on the first test rather than in a constructor. The store and
// the durability stub are INJECTED the way a composition root injects them, so
// these tests drive the same surface MAIN does.
METHOD PRIVATE _M_Arm
IF _init THEN
    RETURN;
END_IF
_init := TRUE;
_u.Setup(Name := 'Test.Durability');
_u();
_u.SetConfigStore(Store := _store);
_u.SetConfigPersistence(Provider := _persist);
// Not under test here: a volatile table, so no previous run's file is a precondition.
_users.M_UseKey(Key := '');
_users.Register(User := 'eng', Pin := '4242', Level := E_AccessLevel.ENGINEER);
_u.Access.Setup(Provider := _users, pAlarmLog := ADR(_u.AlarmLog));
END_METHOD

// Take every outstanding restore loss from the root, exactly as OnCyclic does,
// and leave the LAST one in the suite's fields.
METHOD PRIVATE _M_TakeLoss : BOOL
VAR
    guard    : INT;
    path     : STRING(80);
    expected : UINT;
    found    : UINT;
END_VAR
_M_TakeLoss := FALSE;
FOR guard := 1 TO 8 DO
    // Outputs are written whatever the call returns, so binding the suite's
    // fields directly let the terminating FALSE call blank the loss it had
    // just taken. Take into locals; keep only a take that succeeded.
    IF NOT _u.M_TakeRestoreLoss(Path => path, Expected => expected,
            Found => found) THEN
        RETURN;
    END_IF
    _path := path;
    _expected := expected;
    _found := found;
    _M_TakeLoss := TRUE;
END_FOR
END_METHOD

METHOD First_boot_initializes_silently
TEST('First_boot_initializes_silently');
_M_Arm();
_M_TakeLoss();                            // clear anything an earlier test left
_version := 0;                            // never written
AssertFalse(Condition := _u.Child.M_RestoreStationCfg(pVersion := ADR(_version),
    SchemaVersion := 1),
    Message := 'a first boot has no values to restore, so the caller defaults');
AssertEquals_UINT(Expected := 1, Actual := _version,
    Message := 'the version is stamped forward, so the next boot is an ordinary restore');
AssertFalse(Condition := _M_TakeLoss(),
    Message := 'a first boot LOST nothing and shall not annunciate (3.8b)');
TEST_FINISHED();
END_METHOD

METHOD A_matching_version_restores_and_reports_nothing
TEST('A_matching_version_restores_and_reports_nothing');
_M_Arm();
_M_TakeLoss();
_version := 1;
AssertTrue(Condition := _u.Child.M_RestoreStationCfg(pVersion := ADR(_version),
    SchemaVersion := 1),
    Message := 'a recognized image restores, and the caller keeps its values');
AssertFalse(Condition := _M_TakeLoss(),
    Message := 'a successful restore reports nothing');
TEST_FINISHED();
END_METHOD

